  iR_VacuumAnalogMinDigit                   : UINT := 0;      (*Min value analog-input in digit*)
  iR_VacuumAnalogMaxDigit                   : UINT := 32737;  (*Max value analog-input in digit*)
  fR_VacuumAnalogMinMBar                    : REAL := 0;      (*Min value analog-input in mBar*)
  fR_VacuumAnalogMaxMBar                    : REAL := 50.0;   (*Max value analog-input in mBar*)
  fR_VacuumWarningLevelMBar                 : REAL := 20.0;   (*Warning level in mBar*)
  fR_VacuumErrorLevelMBar                   : REAL := 10.0;   (*Error level in mBar*)

  iR_ParticleMeasurementWarning             : INT := 40;      (*Particle measurement warning level*)
END_VAR

VAR CONSTANT
  iC_ParticleMeasurementNb                  : INT := 60;      (*Number of particle measurements*)
END_VAR

bO_FUReady := bI_FUReady;

fb_TofFUOffDelay(IN := bI_PrintActive, PT := tR_FUOffDelay);
bO_FUActivate := fb_TofFUOffDelay.Q;

fL_VacuumAnalogLevelMBar := UINT_TO_REAL(iI_VacuumMeasurement) * fR_VacuumAnalogMaxMBar / iR_VacuumAnalogMaxDigit;
  
fb_TonVacuumCheckDelay(IN := bO_FUActivate, PT := tR_VacuumCheckDelay);
IF fb_TonVacuumCheckDelay.Q THEN
  (*Level detection for messaging*)
  bO_VacuumWarningLevel := fL_VacuumAnalogLevelMBar < fR_VacuumWarningLevelMBar;
  bO_VacuumErrorLevel   := fL_VacuumAnalogLevelMBar < fR_VacuumErrorLevelMBar;
END_IF

AerosolMeasurement();

ACTION AerosolMeasurement:
fb_RTrigDataReceived(CLK := bI_AerosolMeasurementDataRec);
fb_FTrigDataReceived(CLK := bI_AerosolMeasurementDataRec);

CASE iL_COMstate OF
0:
  IF NOT bI_AerosolMeasurementAckInit THEN
    bO_AerosolMeasurementReqInit := TRUE;
  ELSE
    bO_AerosolMeasurementReqInit := FALSE;

    iL_COMstate := 1;

    bO_AerosolMeasurementAckRec := bI_AerosolMeasurementDataRec;
  END_IF

1:	(*Receive data*)
  IF    fb_RTrigDataReceived.Q
     OR fb_FTrigDataReceived.Q 
  THEN
    bO_AerosolMeasurementAckRec := bI_AerosolMeasurementDataRec;

    cL_Value := iI_AerosolMeasurementRecDataLength;

    aL_ReceivedData := '';
    FOR iL_Counter := 0 TO (cL_Value - 2) DO  (*Without Suffix*)
      aL_ReceivedData := CONCAT(aL_ReceivedData, F_ToCHR(cI_AerosolMeasurementRxBuff[iL_Counter]));
    END_FOR

    iL_ReceiveCount := iL_ReceiveCount + 1;
  END_IF

  IF    bI_AerosolMeasurementBufferFull
     OR bI_AerosolMeasurementFramingError
     OR bI_AerosolMeasurementOverRunError
  THEN
    iL_COMstate := 666;
  ELSE
    eO_ComState := eOpen;
  END_IF

666:	 (* ERROR STATE*)
  eO_ComState := ePortFaulty;	(*ERROR system*)
  iL_COMstate := 0;

END_CASE

fb_TonMeasurementTrigger(IN := NOT fb_TonMeasurementTrigger.Q, PT := T#10S);
IF fb_TonMeasurementTrigger.Q AND bO_FUActivate THEN
  fL_ParticleMeasurements[iL_ParticleMeasurementIdx] := fL_VacuumAnalogLevelMBar; (*TEST with fL_VacuumAnalogLevelMBar !!!*)
  iL_ParticleMeasurementIdx := iL_ParticleMeasurementIdx + 1;
  
  IF iL_ParticleMeasurementIdx > iC_ParticleMeasurementNb THEN
    FOR iL_Counter := 2 TO iC_ParticleMeasurementNb DO
      fL_ParticleMeasurements[iL_Counter - 1] := fL_ParticleMeasurements[iL_Counter];
    END_FOR
    iL_ParticleMeasurementIdx := iC_ParticleMeasurementNb;
  END_IF
END_IF
END_ACTION

METHOD mAckError : BOOL
VAR_INPUT
END_VAR
bO_VacuumWarningLevel := FALSE;
bO_VacuumErrorLevel   := FALSE;
END_METHOD

END_FUNCTION_BLOCK

// ---- POUs/Projects/Print/PRG_PRINT.TcPOU
PROGRAM PRG_PRINT
(*************************************************************************************************)
(*  FILENAME:    PRG_PRINT.EXP                                                                   *)
(*  PROJECT:     CALMAR PUPLC                                                                    *)
(*  COPYRIGHT:   All rights reserved (c) Wifag//Polytype, Fribourg/Switzerland (2016)            *)
(*  ENVIRONMENT: TwinCAT PLC                                                                     *)
(*  VERSION:     <version>                                                                       *)
(*************************************************************************************************)
(*  DESCRIPTION:                                                                   <description> *)
(*    Controls the digital print system.                                                         *)
(*    Main functions: start detection, printhead master, print unit, print group, print          *)
(*    controller.                                                                                *)
(*                                                                                </description> *)
(*************************************************************************************************)

VAR_INPUT
  (*EL5101*)
  lIKp_EncPulse                       AT%I* : ARRAY [1..iCPr_NB_PM] OF UDINT;       (*current encoder position*)
  bI_EncoderWcState                   AT%I* : ARRAY [1..iCPr_NB_PM] OF BOOL;        (*EL5101 encoder WcState*)
  
  bI_PuStopByInk                            : BOOL;  // PU stop and lock start from ink system
END_VAR

VAR_OUTPUT
  (*Interface OUT to PRG_INK / PRG_MACHINE*)
  bO_InitOk                                 : BOOL := FALSE;  (*Init Ok*)
  bO_PrintSystemOk                          : BOOL := TRUE;
  bO_TemperatureOk                          : BOOL := TRUE;
  bO_TotalWcState                           : BOOL := FALSE;  (*Monitoring: WcStates from all terminals*)
END_VAR

VAR
  nCtr, nCtr2 : UDINT;
  
  // ADS interface instances & mapping and responsible FBs
  // -------------------------------------------------------------
  FB_PU                                     : ARRAY [1..iCPr_NB_PU] OF FB_PU;               (*PU - Print Unit*)
  sAdsPrintUnit                             : ARRAY [1..iCPr_NB_PU] OF ST_ADS_PU;
  sL_BLK_PU                                 : ARRAY [1..iCPr_NB_PU] OF ST_MAP_BLK;
  sPuSettings                               : ST_PuSettings;                            // FB_PU configuration
  
  (*{attribute 'TcLinkTo' := '
    [1].fbPrintPosition.IlEncoderPulse := TIIB[RiGen5_v2]^Input^dsfsdfsa;
  '}*)
  fbPrintModule                             : ARRAY [1..iCPr_NB_PM] OF FB_PrintModule_WEU;
  sAdsPrintModule                           : ARRAY [1..iCPr_NB_PM] OF ST_ADS_PM;           (*PM -  Print Module *)
  sL_BLK_PM                                 : ARRAY [1..iCPr_NB_PM] OF ST_MAP_BLK;
//FB_PG                                     : ARRAY [1..iCPr_NB_PG] OF FB_PG;               (*PG -  Print Group *)
  sAdsPrintGroup                            : ARRAY [1..iCPr_NB_PG] OF ST_ADS_PG;
  sL_BLK_PG                                 : ARRAY [1..iCPr_NB_PG] OF ST_MAP_BLK;
  FB_PC                                     : ARRAY [1..iCPr_NB_PC] OF FB_PC;               (*PC - Print Controller*)
  sAdsPrintController                       : ARRAY [1..iCPr_NB_PC] OF ST_ADS_PC;
  sL_BLK_PC                                 : ARRAY [1..iCPr_NB_PC] OF ST_MAP_BLK;
  pFB_PC                                    : POINTER TO ARRAY [1..iCPr_NB_PC] OF POINTER TO FB_PC;
  //pFB_PC                                    : ARRAY [1..iCPr_NB_PC] OF POINTER TO FB_PC;    (* pointer array to PCs*)
  FB_PH                                     : ARRAY [1..iCPr_NB_PH] OF FB_PH_Grid;          (*PH - Print Head*)
  sAdsPrintHead                             : ARRAY [1..iCPr_NB_PH] OF ST_ADS_PH;
  sL_BLK_PH                                 : ARRAY [1..iCPr_NB_PH] OF ST_MAP_BLK;
  sAdsSheetAlignment                        : ARRAY [1..iCPr_NB_PU] OF ST_ADS_DVTSHEETALIGNMENT;          (*SA - Sheet alignement*)
  sL_BLK_SA                                 : ARRAY [1..iCPr_NB_PU] OF ST_MAP_BLK;
  sAdsSubstrate                             : ARRAY [1..iCPr_NB_SUBSTRATE_DEVICES] OF ST_ADS_SUBSTRATE;   (*SUB - Substrate*)
  sL_BLK_SUB                                : ARRAY [1..iCPr_NB_SUBSTRATE_DEVICES] OF ST_MAP_BLK;
  sAdsCamera                                : ARRAY [1..iCPr_NB_PU] OF ST_ADS_CAMERA;                     (*CAM - Camera*)  
  sL_BLK_CAMERA                             : ARRAY [1..iCPr_NB_PU] OF ST_MAP_BLK;          (*array of all camera blocks information*)
  // -------------------------------------------------------------

  // -------------------------------------------------------------
  // Configuration
  sC_Ads_Info                               : ST_ADS_INFO;      // PRG information for ADS block manager
  sMappingInfo                              : T_MapInfo;        // Block mapping configuration
  ISystemBase                               : I_SystemBase;     // reference to system base
  iSystemStatus                             : I_SystemStatus;   // System status interface
  //iSystemCmd                                : I_SystemCmd;      // System interface command
  
  pModuleDef                                : POINTER TO FB_ModuleDef;    // Module definition in system
  sC_Config_P                               : ST_CONFIG_P;      // PRG configuration  
  bL_InitRemVar                             : BOOL := TRUE;
  
  fbModuleMaster                            : FB_ModuleMaster;

  fbPm                                      : FB_ProdManager_DMAX;
  fbHardwarePool                            : FB_HardwarePool;
  fbDefGridParamMediator                    : FB_DefGridParamMediator;
     

  fbWorkerInspection                        : FB_WorkerDefGrid_Inspection;
  fbWorkerVerify                            : FB_WorkerDefGrid_Verify;
  fbWorkerDelete                            : FB_WorkerDefGrid_Delete;
  
  // globals
  rtPuStop                                  : R_TRIG;
  fbOd                                      : FB_OD;        // CoE object dictionary
  
  iWorker                                   : I_Worker;
  
  
  (* --- Maintainance variables ---*)
  (* - file download - *)
  (* -- fw/hw upgrade -- *)
  //fb_fwhw_update                            : FB_CALMAR_UPDATE;
	(* -- hib remote update -- *)
	//fb_pc_hib_rupd                            : ARRAY[1..iCPr_NB_PC] OF FB_PC_HIB_RUPD;(*HIB remote update channels*)
  //fb_hib_rup                                : FB_HIB_UPDATE;                         (*HIB remote updater*)
  (* -- stiching mask manager -- *)
  fb_fdl_mask                               : FB_FILE_DOWNLOAD;                      (*Mask file downloader*)
  (** -- waveform manager -- *)
  fb_fdl_waveform                           : FB_FILE_DOWNLOAD;                      (*waveform file downloader*)
  bWaveformDownloadErr                      : BOOL;                                  (*a waveform douwnload exitst (needed in RIGEN5 only)*)
  tOn_waveform                              : ARRAY[1..iCPr_NB_PC] OF TON;
  bL_waveform_request                       : ARRAY[1..iCPr_NB_PC] OF BOOL;
  lL_PhActStoragetankAssignmentIndex        : ARRAY[1..iCPr_NB_PH] OF DINT;
  lL_MemPhActStoragetankAssignmentIndex     : ARRAY[1..iCPr_NB_PH] OF DINT;
  
  

  
  
  
  
 (*----- Inspection System -----*)
  //bInspectionTrigger : BOOL;
  //fbInspectionSystemTrigger                 : FB_InspectionSystemTrigger;   // Inspection system trigger 
  //nInspectionSystemMarkIdx                  : INT := 3;

  // Neutral fibre calculation with additional mark sensors
  fbNeutralFibreDetermine                   : FB_NeutralFibreDetermine;    // Neutral fibre determine 
    
  (*----- Messages -----*)
  fb_Msg                                    : ARRAY [1..iC_NUM_MSG] OF FB_MESSAGE; (*global Module messages*)
  
  (* -- Recipe read/write auto-management*)
  pFbRecipeMngr                             : POINTER TO FB_RECIPE_READ_WRITE;
  
 
  
  (*----- print, offfset and motion variables ------*)
  // Trigger & Offsets
  //bL_StartTrigger                           : ARRAY [1..iCPr_NB_PM] OF BOOL;       (*Start Trigger for X0*)
  //rT_StartTrigger                           : ARRAY [1..iCPr_NB_PM] OF R_TRIG;
  nL_X0                                     : ARRAY [1..iCPr_NB_PM] OF DINT;       (*detected X0 position*)
  nL_X0_Comp                                : ARRAY [1..iCPr_NB_PM] OF DINT;       (*detected & adapted X0 start position*)
  nL_XS                                     : ARRAY [1..iCPr_NB_PG] OF DINT;       (*Shifted position of start print in pulse*)


  {warning 'TODO: refactor usage in PRG_INK'}
  stPcFlags                                 : ARRAY[1..iCPr_NB_PG] OF CalmarCompPrint.ST_PC_FLAGS;

  // Print module synchronisation
  //fbModuleSynchronisation                   : FB_ModuleSynchronisation;
  //bL_DisableModuleSynchronisation           : BOOL;   (*Visu: disable ModuleSynchronisation*)
  
  
  (*View*)
  // - VISU_SERVICE
  nServiceVisuFrameIndex                    : UINT := 0;   // VISU_SERVICE frame selection
  fbPrintOverview                           : FB_PrintOverview;
  
  (*Debug & Insight*)
  fbPrgPrintTest                            : FB_PrgPrint_test;
  LogPrSetup                                : T_NamedBase;  // just a I_LogSourceMacro implementation (logging PRINT module setup things)
  ePrint_LogLevel                           : E_LogSeverity  := E_LogSeverity.Debug;
  fbProfiler                                : FB_PrgProfiler;

  (*Simulation*)
  bSimulation                               : BOOL;
END_VAR
VAR CONSTANT
  (*Messaging*)
	iC_NUM_MSG                                : INT := 5;
	iC_MSG_1_FOE_MASK_ERR                     : INT := 1;
	iC_MSG_2_FOE_WAVEFORM_ERR                 : INT := 2;
  iC_MSG_3_FOE_CBFW_ERR                     : INT := 3;
  iC_MSG_4_FOE_HIBFW_ERR										: INT := 4;
  iC_MSG_5_PC_SUPPLY_OFF                    : INT := 5;
END_VAR

(* INIT First action init call*)
IF NOT bO_InitOk THEN
  Init();
  RETURN;
END_IF;

(* Call ACTIONS *)
(*************************************************************************************************)
RemVar();           (*Call update remanent data action*)
DownloadFiles();    (*Call file downloads*)
Testing();          (*Call test code*)
fbProfiler();
setLoggingLevels();


// Main/MasterModule part
fbModuleMaster();

// --------------------------------------------------------
// Print Blocks (global for all)
// -- CT and ProdMngr (Production Management)


fbOd();
fbPm();
fbHardwarePool();


// -- PM print modules
FOR nCtr := 1 TO TO_UDINT(iCPr_NB_PM) DO
  
  FOR nCtr2 := 1 TO TO_UDINT(GVL_WEU.nC_WorkerPrintPerPm) DO
    {warning 'TODO: scale X Offset with fL_WebStretchCalculated?'}
    fbPrintModule[nCtr].fPrintOffsetX[nCtr2]       :=  TO_LREAL(sAdsPrintUnit[ePr_PU_UNIT_1].sI_ShiftJobX.lI_Val) / 1_000_000 	// PU [um] to [m]
                                                     + TO_LREAL(sAdsPrintModule[nCtr].sI_GeneralShiftX.lI_Val) / 1_000_000 	  // PG [um] to [m]
                                                     + TO_LREAL(sAdsPrintGroup[nCtr2 + TO_UDINT(iCPr_MAP_PM_PG[nCtr2])-1].sI_ShiftPositionX.lI_Val) / 1_000_000;
    fbPrintModule[nCtr].fPrintOffsetY[nCtr2]       :=  DINT_TO_LREAL(F_MeterToSubPixel(DINT_TO_LREAL(sAdsPrintUnit[ePr_PU_UNIT_1].sI_ShiftJobY.lI_Val ) / 1_000_000, nC_PrintResolution))   (*[um] to [px] job yOffset from upper level (GUI)*)
                                                     + DINT_TO_LREAL(F_MeterToSubPixel(DINT_TO_LREAL(sAdsPrintModule[nCtr].sI_GeneralShiftY.lI_Val )    / 1_000_000, nC_PrintResolution))   (*[um] to [px] job yOffset from upper level (GUI)*)
                                                     + DINT_TO_LREAL(F_MeterToSubPixel(DINT_TO_LREAL(sAdsPrintGroup[nCtr2 + TO_UDINT(iCPr_MAP_PM_PG[nCtr2])-1].sI_ShiftPositionY.lI_Val) / 1_000_000, nC_PrintResolution));   (*[um] to [px] job yOffset from upper level (GUI)*)
                                                      
	END_FOR
    
  fbPrintModule[nCtr]();
END_FOR



// Print module synchronisation (simulation not for production)
(*
fbModuleSynchronisation( IbEnable           := NOT bL_DisableModuleSynchronisation
                       , IbEngaged          := bL_Engaged
                       , IbPrintEnabled     := bL_PrintEnabled
                       , InFormatLength     := nL_FormatLength
                       , InModule2ToModule3 := nL_Module2ToModule3
                       , IbFormatTrig       := bL_StartTrig
                       , ObPrintEnabled     => bL_PrintEnabledSync); 
*)


// --------------------------------------------------------
// Worker chain  --> call all work() methods
iWorker := fbWorkerDelete.Root;
WHILE iWorker <> 0 DO
  iWorker.work();
  iWorker := iWorker.Next;
END_WHILE


(* -- PU PrintUnit*)
// PG->PU status/flags 
FOR nCtr := 1 TO TO_UDINT(iCPr_NB_PU) DO 
  // specific handling
  rtPuStop(CLK := bI_PuStopByInk);       (*If varnish change is activated the job should be stopped.*)
  IF rtPuStop.Q THEN FB_PU[nCtr].reqPuStop('Stop by InkSystem'); END_IF
  
  FB_PU[nCtr]();
  
  // WEU Start CanEx override
  sAdsPrintUnit[nCtr].sI_Start.bO_CommandCanEx := sAdsPrintUnit[nCtr].sI_Start.bO_CommandCanEx 
                                                AND NOT iSystemStatus.bSleep     // sleep active
                                                AND NOT bI_PuStopByInk;          // ink system locks start
END_FOR

// Inspection system
{warning 'TODO: create a worker for inspection system'}
(*
IF (nInspectionSystemMarkIdx > 3) OR (nInspectionSystemMarkIdx < 2) THEN nInspectionSystemMarkIdx := 3; END_IF  (*Index check*)
fbInspectionSystemTrigger.UsePositionTrigger := fbStartPositionSimulationHOA._bSim AND NOT bL_DisableSimMarkStartTriggerM3;
(*input bI_SensorState depends on _bUsePositionTrigger*)
IF fbInspectionSystemTrigger.UsePositionTrigger THEN
  fbInspectionSystemTrigger.bI_SensorState := bMasterTrigger;
ELSE
  fbInspectionSystemTrigger.bI_SensorState := Fb_PaperPosDetect[nInspectionSystemMarkIdx - 1].bIKp_StartSensor;
END_IF

fbInspectionSystemTrigger.bI_SensorState
fbInspectionSystemTrigger( iI_CurrentPos         := nMasterPosition
                         , fI_ConveyorSpeed      := fMasterSpeed
                         , iI_SensorX0           := SEL(bL_Engaged[1], nL_X0[2]                           , nL_X0[1])
                         , tI_SensorTimeStampPos := Fb_PaperPosDetect[nInspectionSystemMarkIdx - 1].tIKp_TimeStampPos
                         (*StartTrigger Simulation VISU&FB*)
                       //, bI_ManualTrigger      := fbStartPositionSimulation.bStartTrig
                         );
*)

// Neutral fibre calculation with additional mark sensors
fbNeutralFibreDetermine(fSpeed := fbModuleMaster.fMasterSpeed);


(*--- VISU stuff ----------------*)
// fix offset (left visu border) + VerifyWorker = a constant position => calculate a pixel to m ratio
fbPrintOverview.fX_m  := fbWorkerDelete.fPosition; // (0.2 + fbWorkerVerify.fWorkerToMasterRef) + fbModuleMaster.fLastModuleOffset + (fbModuleMaster.fDetectToRefPos);
fbPrintOverview.fY_m  := 2;
fbPrintOverview.nX_px := 800;
fbPrintOverview.nY_px := 300;
fbPrintOverview.fPxToMRatio := fbPrintOverview.nX_px / fbPrintOverview.fX_m;
fbPrintOverview.iPrintPosition := fbModuleMaster.iMasterPrintPosition;

fbPrintOverview();
(*------------------------------*)

(****************************************************************************)
(* Messaging, NOTE: they are using the FB_PU message handler! *)
(* ------------------------------------------------------------------------ *)
fb_Msg[iC_MSG_1_FOE_MASK_ERR]    .bI_Status := fb_fdl_mask.bO_Error;
fb_Msg[iC_MSG_2_FOE_WAVEFORM_ERR].bI_Status := FALSE;  //bWaveformDownloadErr; // fb_fdl_waveform.bO_Error;
fb_Msg[iC_MSG_3_FOE_CBFW_ERR]    .bI_Status := fbHardwarePool.bError_fwhw_update;
fb_Msg[iC_MSG_4_FOE_HIBFW_ERR]   .bI_Status := fbHardwarePool.bError_hib_rup;
fb_Msg[iC_MSG_5_PC_SUPPLY_OFF]   .bI_Status := FALSE; //TODO: NOT PRG_MACHINE.sL_CvyrStatus.bI_PowerState;

FOR nCtr := 1 TO TO_UDINT(iC_NUM_MSG) DO
  IF fb_Msg[nCtr].pI_MsgConfig <> 0 AND fb_Msg[nCtr].iI_MsgNumber <> 0 THEN
    fb_Msg[nCtr]();
  END_IF
END_FOR 

(****************************************************************************)
(* Global states *)
(* ------------------------------------------------------------------------ *)
bO_PrintSystemOk := fbPm.bReady;
(*WcState: 0 = Data valid, 1 = Data invalid*)
bO_TotalWcState :=    bI_EncoderWcState[1]
                   OR bI_EncoderWcState[2];

METHOD DownloadFiles
VAR
  lCtr : INT;
  sPcFlags : ST_PC_FLAGS;
  aDefaultWaveform : T_MaxString;
  aInkWaveform : T_MaxString;
END_VAR
(* PC firmware updater*)
(*    uses PC[x] FoE channel *)
(* ------------------------------------------------------------------------ *)
(* --- START: --- *)
//fb_fwhw_update( pI_fbPc := pFB_PC^);
(* --- END: --- *)


(****************************************************************************)
(* HIB remote update*)
(*    uses PC[x] FoE channel *)
(* ------------------------------------------------------------------------ *)
(* --- START: --- *)
//fb_hib_rup();
(* --- END: --- *)


(****************************************************************************)
(* mask update*)
(*		uses PC[x] FoE channel *)
(* ------------------------------------------------------------------------ *)
(* --- START: printhead mask loader --- *)
(*FOR lCtr := 1 TO iCPr_NB_PC DO
  IF FB_PC[lCtr].sO_PcFlags.bBoardEnterOp THEN 
    fb_fdl_mask.Start(DINT_TO_INT(lCtr));    // start individual channel
	END_IF
END_FOR;*)
fb_fdl_mask();
(* --- END: printhead mask loader --- *)


(****************************************************************************)
(* Waveform update*)
(*    uses PC[x] FoE channel *)
(* ------------------------------------------------------------------------ *)
(* --- START: printhead waveform loader --- *)
bWaveformDownloadErr := FALSE;
FOR lCtr := 1 TO iCPr_NB_PC DO
  sPcFlags := FB_PC[lCtr].sPcFlags;
  bL_waveform_request[lCtr] := tOn_waveform[lCtr].Q;
  IF    ( sPcFlags.bBoardEnabling ) 
     OR ( bL_waveform_request[lCtr] ) //filtered internally: AND NOT fb_fdl_waveform[iL_Counter].bO_Busy AND (tTimeoutWavef[iL_Counter].Q OR fb_Wavef_CfgTrig[iL_Counter].Q)
  THEN
    fb_fdl_waveform.Start(DINT_TO_INT(lCtr));    // start individual channel
  END_IF

  tOn_waveform[lCtr](IN:=sPcFlags.bWaveform AND NOT bL_waveform_request[lCtr], PT:= T#14S);

  // build global request for message
  IF sPcFlags.bWaveform AND FB_PC[lCtr].bBoardEnable THEN 
    bWaveformDownloadErr := TRUE;
	END_IF
END_FOR;
fb_fdl_waveform();

(*Assign WaveFileName from storage tank to PH. Trigger transmit of waveform if new name is set.*)
FOR lCtr := 1 TO iCPr_NB_PH DO
  lL_PhActStoragetankAssignmentIndex[lCtr] := PRG_INK.iL_ActStoragetankAssignmentIndex[iCPr_MAP_PH_HT[lCtr]];

  (*If lL_PhActStoragetankAssignmentIndex is assigned to a storage tank the waveform must be copied.*)
  IF     (lL_PhActStoragetankAssignmentIndex[lCtr] > 0)
     AND (lL_PhActStoragetankAssignmentIndex[lCtr] <> lL_MemPhActStoragetankAssignmentIndex[lCtr])
  THEN
    // set new waveform name to PH
    aDefaultWaveform := fb_fdl_waveform.aI_src_file_name_default;
    aInkWaveform := PRG_INK.sAdsIkInkStorageTank[lL_PhActStoragetankAssignmentIndex[lCtr]].sI_InkParameter.aWaveform; 
    
    IF aInkWaveform <> '' AND aInkWaveform <> 'undef' AND aInkWaveform <> 'undef.wav' THEN  // use only when waveform from storage assignemen is ok, else keep ph ads value
      sAdsPrintHead[lCtr].aI_WaveFileName := PRG_INK.sAdsIkInkStorageTank[lL_PhActStoragetankAssignmentIndex[lCtr]].sI_InkParameter.aWaveform;      
		END_IF

    (*Fix extension if not existing in the file name*)
    IF (FIND(sAdsPrintHead[lCtr].aI_WaveFileName, '.wav') = 0) AND (FIND(sAdsPrintHead[lCtr].aI_WaveFileName, '.WAV') = 0) THEN
      sAdsPrintHead[lCtr].aI_WaveFileName := CONCAT(sAdsPrintHead[lCtr].aI_WaveFileName, '.wav');
    END_IF

    (*check for valid file name*)
     IF sAdsPrintHead[lCtr].aI_WaveFileName = 'undef.wav' OR sAdsPrintHead[lCtr].aI_WaveFileName = '.wav' OR sAdsPrintHead[lCtr].aI_WaveFileName = '' THEN
       LogPrSetup.LogError(F_Concat5('Invalid waveform filename: ', sAdsPrintHead[lCtr].aI_WaveFileName, ' on PH[', TO_STRING(lCtr),']'));
       sAdsPrintHead[lCtr].aI_WaveFileName := aDefaultWaveform;
       LogPrSetup.LogError(F_Concat5('Set default waveform filename: ', sAdsPrintHead[lCtr].aI_WaveFileName, ' on PH[', TO_STRING(lCtr),']'));
		 END_IF
  END_IF

  lL_MemPhActStoragetankAssignmentIndex[lCtr] := lL_PhActStoragetankAssignmentIndex[lCtr];
END_FOR
END_METHOD

METHOD Init : BOOL
VAR
  nCtr : UDINT;
  nPhCtr : UDINT;
  pAdsPg : ARRAY[1..GVL_WEU.nC_WorkerPrintPerPm] OF POINTER TO ST_ADS_PG;
END_VAR
(*************************************************************************************************)
(* --- Module preprarations --- *)

// Get system reference
IF ISystemBase = 0 THEN
  ISystemBase := PRG_SYSTEMBASE.getSystemBaseInterface();
  IF ISystemBase = 0 THEN 
    RETURN; 
  END_IF
END_IF

// Wait until system(base) is booted
IF ISystemBase.bBooting THEN RETURN; END_IF
PRG_SYSTEMBASE.getSystemStatusInterface(iSystemStatus=>iSystemStatus);
//PRG_SYSTEMBASE.getSystemCmdInterface(iSystemCmd=>iSystemCmd

// Build mapping information for ADS
Mapping();

// Register module to system
pModuleDef := ISystemBase.regModule(
  pAdsInfo := ADR(sC_Ads_Info),
  pMapInfo := ADR(sMappingInfo)
);
IF pModuleDef = 0 THEN RETURN; END_IF

// remanent init 
RemVar();



(*************************************************************************************************)
(* Init FB and ADS instances*)
setLoggingLevels();

(*-- Print blocks init --------------------------------------------------------------------------*)
(*-- Module Master*)
fbModuleMaster.Init(pPU:=ADR(FB_PU[1]), pProdMngr:=ADR(fbpm), iHwPool:=fbHardwarePool);


(*-- CoE object dicionary*)
fbOd.init(aAmsNetId:=sC_AMSNETID_LOCALHOST, aFilePath:=F_Concat3(aC_PlcConfigPath, aC_PlcFlashFileSubPath, 'od.json'), pSimString:=0);

(* -- PU PrintUnit*)
FOR nCtr := 1 TO TO_UDINT(iCPr_NB_PU) DO
	(*-- ADS --*)
  setupAdsPu(pAds:=ADR(sAdsPrintUnit[nCtr]), nIdx:=nCtr);
  setupAdsSa(pAds:=ADR(sAdsSheetAlignment[nCtr]));
  
	(*-- FB --*)
  sPuSettings.bStopAfterDone := FALSE;
  FB_PU[nCtr].Init(                                                  (*Init referenced & config for FB*)
                    pAdsIf        := ADR(sAdsPrintUnit[nCtr])        (*> ads pu reference*)
                  , pAdsSubstrate := ADR(sAdsSubstrate[1])           (*> ads substrate ref*)
                  , pPuSettings   := ADR(sPuSettings)
                  , iNumPg        := iCPr_NB_PM                      (*> Number print SubSystems*)
                  );
END_FOR;


(* -- PG PrintGroup*)
FOR nCtr := 1 TO TO_UDINT(iCPr_NB_PG) DO
	(*-- ADS --*)
  setupAdsPg(pAds:=ADR(sAdsPrintGroup[nCtr]), nIdx:=nCtr);

  (*-- IF direct access to PRG_INK --*)
  PRG_INK.pAdsPg[nCtr] := ADR(sAdsPrintGroup[nCtr]);  
END_FOR;


// !!! Init HW before module (PCs, PHs) !!! --------------------
(* -- PC Print Controller*)
FOR nCtr := 1 TO TO_UDINT(iCPr_NB_PC) DO
	(*-- PC --*)
	FB_PC[nCtr].Init( pAds               := ADR(sAdsPrintController[nCtr])
                  , sAmsNetIdLocalHost := sC_AMSNETID_LOCALHOST
                  , sAmsNetIdIo        := sC_AMSNETID_IO
                  , nEcatSlaveAddr     := iG_PC_ADDRESS[nCtr]
                  , nBlockId           := ePr_BLK_PC
                  , pOd                := ADR(fbOd)
                  , tWaveDownload      := T#10S
                  );
  
  // hw enable inputs not existing -> enable initially
  FOR nPhCtr := 1 TO TO_UDINT(iCPr_NB_PH_PER_CONTROLLER) DO
    FB_PC[nCtr].bI_PhHwEnable[nPhCtr] := TRUE;
  END_FOR

	(*-- ADS --*)
  setupAdsPc(pAds:=ADR(sAdsPrintController[nCtr]), nIdx:=nCtr);
END_FOR;


(*PH - Print Head*)
FOR nCtr := 1 TO TO_UDINT(iCPr_NB_PH) DO
	(*-- ADS --*)
  setupAdsPh(pAds:=ADR(sAdsPrintHead[nCtr]), nIdx:=nCtr);
     
  fbPrintModule[iCPr_PH_MAPPING[nCtr].nPm].RegisterHw(
    pPc:=ADR(FB_PC[iCPr_PH_MAPPING[nCtr].nPcInst]),
    pPh:=ADR(FB_PH[iCPr_PH_MAPPING[nCtr].nPhInst]),
    pMapDef:=ADR(iCPr_PH_MAPPING[nCtr])
  );

  (*-- PH --*)
  FB_PH[nCtr].init( pAdsIf       := ADR(sAdsPrintHead[nCtr])
                  , sPhDef       := GVL_PrintDef.RIGEN5
                  , tTempMonitor := T#45S
                  );
END_FOR;


(*----SUBSTRATE init*)
FOR nCtr := 1 TO TO_UDINT(iCPr_NB_SUBSTRATE_DEVICES) DO
  setupAdsSub(pAds:=ADR(sAdsSubstrate[nCtr]), nIdx:=nCtr); 
END_FOR


(*-- PrintModules*)
FOR nCtr := 1 TO TO_UDINT(iCPr_NB_PM) DO

	(*-- ADS --*)
  setupAdsPm(pAds:=ADR(sAdsPrintModule[nCtr]), nIdx:=nCtr);
  
  pAdsPg[1] := ADR(sAdsPrintGroup[iCPr_MAP_PM_PG[nCtr]]);
  pAdsPg[2] := ADR(sAdsPrintGroup[iCPr_MAP_PM_PG[nCtr]+1]);
  
  (*-- FB -- *)
  {warning 'TODO: set size: fPrintUnitWidth'}
  fbPrintModule[nCtr].Init( nIdx     := TO_UDINT(nCtr)
                          , pAdsPm   := ADR(sAdsPrintModule[nCtr])
                          , pAdsSa   := ADR(sAdsSheetAlignment[ePr_PU_UNIT_1])
                          , pAdsCam  := ADR(sAdsCamera[1])
                          , pAdsPg   := pAdsPg
                          , fCycleTime := pModuleDef^.fCycleTime_s
                          , fPrintUnitWidth := 1  {warning 'TODO: used for Grid ImageShift somehow and banana correction'}
                          , nYShiftPcCenter := nC_YShiftOffset
                          , iModuleMaster := fbModuleMaster
                          , iPosition := 0  // set internally
                          , iStartPos := 0  // set internally
                          , iSystemStatus := iSystemStatus
                          , pMachineInputs := ADR(PRG_MACHINE.fbMachineComm.sModuleMachineState[nCtr])
                          , pMachineOutputs := ADR(PRG_MACHINE.fbMachineComm.sModuleMachineFeedback[nCtr])
  );
  // register to master
  fbModuleMaster.registerModule(pModule:=ADR(fbPrintModule[nCtr]));
END_FOR;
fbModuleMaster.setMasterModule(ADR(fbPrintModule[1]));


(*-- Print management init ------------------------------------------------------------------*)
fbPm.LogLevel := ePrint_LogLevel;
fbPm.init( pPU    := ADR(FB_PU[ePr_PU_UNIT_1]) 
         , pAdsPU := ADR(sAdsPrintUnit[ePr_PU_UNIT_1]),
         );
fbPm();  // call it once for self-initialisation
FB_PU[ePr_PU_UNIT_1].registerStatusClient(sClient := fbPm);


(*-- Worker init --------------------------------------------------------------------------------*)


// -- Worker Print
//  -> defined in Module

// -- Verify
fbWorkerVerify.Init(iWorkerParams:=fbModuleMaster.iWorkerParams, pMsgConfig:=FB_PU[1].pO_MsgConfig, fPrintResolution := nC_PrintResolution, fSubPxResolution := nC_SubPixelResolution);
fbWorkerVerify.InitWorkerVerify(pPm:=ADR(fbPm));
fbWorkerVerify.reg();
fB_PU[ePr_PU_UNIT_1].registerStatusClient(sClient:=fbWorkerVerify);

// -- Inspection
fbWorkerInspection.Init(iWorkerParams:=fbModuleMaster.iWorkerParams, pMsgConfig:=FB_PU[1].pO_MsgConfig, fPrintResolution := nC_PrintResolution, fSubPxResolution := nC_SubPixelResolution);
fbWorkerInspection.reg();
fB_PU[ePr_PU_UNIT_1].registerStatusClient(sClient:=fbWorkerInspection);

// -- Delete
fbWorkerDelete.Init(iWorkerParams:=fbModuleMaster.iWorkerParams, pMsgConfig:=FB_PU[1].pO_MsgConfig, fPrintResolution := nC_PrintResolution, fSubPxResolution := nC_SubPixelResolution);
fbWorkerDelete.reg();
fB_PU[ePr_PU_UNIT_1].registerStatusClient(sClient:=fbWorkerDelete);


(*-- Camera init ----------------------------------------------------*)

// -- No camera (SheetDetect only)
//fbNoCamera.Init(nPrintUnitResolution:=nC_PrintResolution, nPrintUnitSubPx:=nC_SubPixelResolution, iCameraTrigger:=fbMarkDetection, bUseCameraTrigger:=FALSE, bUseCameraTriggerFeedback:=FALSE);
//fbWorkerCamera.RegisterCamera(fbNoCamera);


// -- Param mediator between Workers
//fbDefGridParamMediator.init(pCreateWorker:=ADR(fbWorkerDefGrid_Python), pCamWorker := ADR(fbWorkerDefGrid_Camera),pDefWorker:= ADR(fbWorkerDefGrid_Deformation));

// register Emergency
(*FOR lCtr := 1 TO iCPr_NB_PG DO
  PRG_SYSTEMBASE.fbEmergency.mRegisterObserver(iObserver := fbWorkerWeu[lCtr]);
END_FOR*)


// Hw Management
//    Hardware Pool for PH - Print Head and PC - Print Controller*)
fBHardwarePool.init(
  sAmsNetIdLocalhost  := sC_AMSNETID_LOCALHOST,
  sAmsNetIdIo         := sC_AMSNETID_IO,
  pOd                 := ADR(fbOd),
  pConfig             := ADR(sC_Config_P)
);
pFB_PC := fbHardwarePool.pPcs;  // used for FileDownload and global FBs managing all PCs




(*************************************************************************************************)
(*FileDownloader*)

//(* - firmware*) - Is now in HardwarePool
//fb_fwhw_update.aI_appl_file_path := F_Concat3(aC_PlcConfigPath, aC_PlcFlashFileSubPath, 'user.appl');
//fb_fwhw_update.aI_fpga_file_path := F_Concat3(aC_PlcConfigPath, aC_PlcFlashFileSubPath, 'user.fpga');
//fb_fwhw_update( pI_fbPc := pFB_PC^);
//fb_fwhw_update.init();

//(* - hib remote upfate*) - Is now in HardwarePool
//fb_hib_rup.bI_Enable   := TRUE;
//fb_hib_rup.aI_FilePath := F_Concat3(aC_PlcConfigPath, aC_PlcFlashFileSubPath, 'user.hib');
//fb_hib_rup( sI_Ary_Fb:=fb_pc_hib_rupd, pI_Ary_Fb_Pc:=pFB_PC^);


(*-- Mask file*)
fb_fdl_mask.bI_Enable                := TRUE;
fb_fdl_mask.aI_src_file_path         := CONCAT(aC_PlcConfigPath, aC_PlcMaskFileSubPath);
fb_fdl_mask.aI_src_file_name_default := 'mask.msk';
fb_fdl_mask.aI_dest_file_path        := 'mask.msk.msk';
FOR nCtr := 1 TO TO_UDINT(iCPr_NB_PC) DO
	FOR nPhCtr := 1 TO TO_UDINT(iCPr_NB_PH_PER_CONTROLLER) DO
		IF iCPr_MAP_PC_PH[nCtr, nPhCtr] <> -1 THEN
	    fb_fdl_mask.aI_src_file_names[nCtr, nPhCtr] := ADR(sAdsPrintHead[iCPr_MAP_PC_PH[nCtr, nPhCtr]].aI_MaskFileName);
		END_IF
	END_FOR
END_FOR
fb_fdl_mask(pI_fbpc:=pFB_PC^);
fb_fdl_mask.Init(
  aDownloaderName := 'Mask downloader',
  bFilePerPh      := TRUE,
  bDefaultFile    := FALSE,
  bShowDetail     := TRUE,
  bUseLock        := FALSE,
  bEnabledOnly    := TRUE,
  bFileNameChange := TRUE,
  bEnterOp        := TRUE,
  bEnabling       := TRUE,
  bUseRange       := FALSE,
  lColorRGB       := 16#FF0080FF,
  iRetryCount     := 0,
  tRetryTimeout   := T#8S,
);

(*-- waveform file*)
fb_fdl_waveform.bI_Enable                := TRUE;
fb_fdl_waveform.aI_src_file_path         := CONCAT(aC_PlcConfigPath, aC_PlcWaveformFileSubPath);
fb_fdl_waveform.aI_src_file_name_default := 'waveform.wav';
fb_fdl_waveform.aI_dest_file_path        := 'waveform.wav.wav';
FOR nCtr := 1 TO TO_UDINT(iCPr_NB_PC) DO
	FOR nPhCtr := 1 TO TO_UDINT(iCPr_NB_PH_PER_CONTROLLER) DO
		IF iCPr_MAP_PC_PH[nCtr, nPhCtr] <> -1 THEN
	    fb_fdl_waveform.aI_src_file_names[nCtr, nPhCtr] := ADR(sAdsPrintHead[iCPr_MAP_PC_PH[nCtr, nPhCtr]].aI_WaveFileName);
		END_IF
	END_FOR
END_FOR
fb_fdl_waveform(pI_fbpc:=pFB_PC^);
fb_fdl_waveform.Init(
  aDownloaderName := 'Waveform downloader',
  bFilePerPh      := FALSE,
  bDefaultFile    := FALSE,
  bShowDetail     := TRUE,
  bUseLock        := FALSE,
  bEnabledOnly    := TRUE,
  bFileNameChange := TRUE,
  bEnterOp        := TRUE,
  bEnabling       := TRUE,
  bUseRange       := FALSE,
  lColorRGB       := 16#FF9191C8,
  iRetryCount     := 0,
  tRetryTimeout   := T#9S,  
);


// View setup
fbPrintOverview.init(
  pCTM:=fbModuleMaster.pCTManager, 
  pWorkerDefGrid:=ADR(fbWorkerDelete)
);

// Inspection system
//fbInspectionSystemTrigger.Init(nResolution := nC_PrintResolution * nC_SubPixelResolution, bUsePositionTrigger := FALSE);

// Neutral fibre calculation with additional mark sensors
fbNeutralFibreDetermine.Init(nResolution := nC_PrintResolution * nC_SubPixelResolution);


(*Messaging*)
(*************************************************************************************************)
(*NOTE: FB_PU[x].init() has to be called before*)
fb_Msg[iC_MSG_1_FOE_MASK_ERR].pI_MsgConfig       := FB_PU[1].pO_MsgConfig;
fb_Msg[iC_MSG_1_FOE_MASK_ERR].iI_MsgLocation     := ePr_BLK_PU;
fb_Msg[iC_MSG_1_FOE_MASK_ERR].iI_MsgNumber       := eCPr_FOE_MASK_DL_ERR;

fb_Msg[iC_MSG_2_FOE_WAVEFORM_ERR].pI_MsgConfig   := FB_PU[1].pO_MsgConfig;
fb_Msg[iC_MSG_2_FOE_WAVEFORM_ERR].iI_MsgLocation := ePr_BLK_PU;
fb_Msg[iC_MSG_2_FOE_WAVEFORM_ERR].iI_MsgNumber   := eCPr_FOE_WAVEFORM_DL_ERR;

fb_Msg[iC_MSG_3_FOE_CBFW_ERR].pI_MsgConfig       := FB_PU[1].pO_MsgConfig;
fb_Msg[iC_MSG_3_FOE_CBFW_ERR].iI_MsgLocation     := ePr_BLK_PU;
fb_Msg[iC_MSG_3_FOE_CBFW_ERR].iI_MsgNumber       := eCPr_FOE_CBFW_DL_ERR;

fb_Msg[iC_MSG_4_FOE_HIBFW_ERR].pI_MsgConfig      := FB_PU[1].pO_MsgConfig;
fb_Msg[iC_MSG_4_FOE_HIBFW_ERR].iI_MsgLocation    := ePr_BLK_PU;
fb_Msg[iC_MSG_4_FOE_HIBFW_ERR].iI_MsgNumber      := eCPr_FOE_HIBFW_DL_ERR;

fb_Msg[iC_MSG_5_PC_SUPPLY_OFF].pI_MsgConfig      := FB_PU[1].pO_MsgConfig;
fb_Msg[iC_MSG_5_PC_SUPPLY_OFF].iI_MsgLocation    := ePr_BLK_PU;
fb_Msg[iC_MSG_5_PC_SUPPLY_OFF].iI_MsgNumber      := eCPr_PC_SUPPLY_OFF;


(*************************************************************************************************)
(* --- System servcices ---- *)
(* -- BlockId saving ----------------------------------------------------------------------------*)
PRG_SYSTEMBASE.fbBlockIdSave.registerModule(
  aI_StoragePath := CONCAT(aC_PlcConfigPath, aC_PlcBlockIdSubPath),
  pI_Ads_Info    := ADR(sC_Ads_Info)
);

// init finished
bO_InitOk := TRUE;

(**** END ****************************************************************************************)
END_METHOD

METHOD Mapping : BOOL
VAR
  lCtr : INT;
END_VAR
(*************************************************************************************************)
(*ADS blocks mapping definition*)
(*************************************************************************************************)
(*mapping of each block with his parents, type and index*)
(*unit -> root*)
sL_BLK_PU[1].iPMaps[1]    := FC_ADD_MAP(eSys_BLK_ROOT, 1);

(*Substrate -> root*)
sL_BLK_SUB[1].iPMaps[1]   := FC_ADD_MAP(eSys_BLK_ROOT, 1);

(*SheetAlignment -> unit*)
sL_BLK_SA[1].iPMaps[1]    := FC_ADD_MAP(ePr_BLK_PU, 1);

(*Camera -> unit*)
sL_BLK_CAMERA[1].iPMaps[1]:= FC_ADD_MAP(ePr_BLK_PU, 1);

(*module*)
FOR lCtr := 1 TO iCPr_NB_PM DO
  (*modules -> unit*)
  sL_BLK_PM[lCtr].iPMaps[1] := FC_ADD_MAP(ePr_BLK_PU, 1);
END_FOR;

(*group*)
FOR lCtr := 1 TO iCPr_NB_PG DO
  (*groups -> module*)
  sL_BLK_PG[lCtr].iPMaps[1] := FC_ADD_MAP(ePr_BLK_PM, iCPr_MAP_PG_PM[lCtr]);
  (*groups -> header tank group*)
  sL_BLK_PG[lCtr].iPMaps[2] := FC_ADD_MAP(eIk_BLK_HEADERTANK_GROUP, iCPr_MAP_PG_HTG[lCtr]);
END_FOR;

(*controller*)
FOR lCtr := 1 TO iCPr_NB_PC DO
  (*controller -> group*)
  IF bCPr_PC_EXIST[lCtr] THEN
    sL_BLK_PC[lCtr].iPMaps[1] := FC_ADD_MAP(ePr_BLK_PG, iCPr_MAP_PC_PG[lCtr]);
  END_IF;
END_FOR;

(*printhead*)
FOR lCtr := 1 TO iCPr_NB_PH DO
  (*printhead -> print controller*)
  IF bCPr_PH_EXIST[lCtr] THEN
    sL_BLK_PH[lCtr].iPMaps[1] := FC_ADD_MAP(ePr_BLK_PC        , iCPr_MAP_PH_PC[lCtr]);
  END_IF;
END_FOR;


(*************************************************************************************************)
(* initialize module information (module and mapping) *)
(*************************************************************************************************)
sC_Ads_Info.bReady   := FALSE;
sC_Ads_Info.aType    := 'PRG_PRINT';
sC_Ads_Info.iVersion := 010000;			(*1.0.0*)
sC_Ads_Info.iType    := eMOD_PRINT;

sMappingInfo.init(lModId:=TO_UINT(eMOD_PRINT));
sMappingInfo.addBlkAry( iAdsBlockType := TO_UINT(ePr_BLK_PU),       aAdsBlockName := 'sAdsPrintUnit',       iAdsBlockVersion:= sAdsPrintUnit[1].iO_Version,                    iNbrBlocks := SIZEOF(sL_BLK_PU)/SIZEOF(sL_BLK_PU[1]),         pBlockArray := ADR(sL_BLK_PU));
sMappingInfo.addBlkAry( iAdsBlockType := TO_UINT(ePr_BLK_PM),       aAdsBlockName := 'sAdsPrintModule',     iAdsBlockVersion:= INT_TO_UINT(sAdsPrintModule[1].iO_Version),     iNbrBlocks := SIZEOF(sL_BLK_PM)/SIZEOF(sL_BLK_PM[1]),         pBlockArray := ADR(sL_BLK_PM));
sMappingInfo.addBlkAry( iAdsBlockType := TO_UINT(ePr_BLK_PG),       aAdsBlockName := 'sAdsPrintGroup',      iAdsBlockVersion:= INT_TO_UINT(sAdsPrintGroup[1].iO_Version),      iNbrBlocks := SIZEOF(sL_BLK_PG)/SIZEOF(sL_BLK_PG[1]),         pBlockArray := ADR(sL_BLK_PG));
sMappingInfo.addBlkAry( iAdsBlockType := TO_UINT(ePr_BLK_PC),       aAdsBlockName := 'sAdsPrintController', iAdsBlockVersion:= INT_TO_UINT(sAdsPrintController[1].iO_Version), iNbrBlocks := SIZEOF(sL_BLK_PC)/SIZEOF(sL_BLK_PC[1]),         pBlockArray := ADR(sL_BLK_PC));
sMappingInfo.addBlkAry( iAdsBlockType := TO_UINT(ePr_BLK_PH),       aAdsBlockName := 'sAdsPrintHead',       iAdsBlockVersion:= INT_TO_UINT(sAdsPrintHead[1].iO_Version),       iNbrBlocks := SIZEOF(sL_BLK_PH)/SIZEOF(sL_BLK_PH[1]),         pBlockArray := ADR(sL_BLK_PH));
sMappingInfo.addBlkAry( iAdsBlockType := TO_UINT(ePr_BLK_SA),       aAdsBlockName := 'sAdsSheetAlignment',  iAdsBlockVersion:= INT_TO_UINT(sAdsSheetAlignment[1].iO_Version),  iNbrBlocks := SIZEOF(sL_BLK_SA)/SIZEOF(sL_BLK_SA[1]),         pBlockArray := ADR(sL_BLK_SA));
sMappingInfo.addBlkAry( iAdsBlockType := TO_UINT(ePr_BLK_SUBSTRATE),aAdsBlockName := 'sAdsSubstrate',       iAdsBlockVersion:= INT_TO_UINT(sAdsSubstrate[1].iO_Version),       iNbrBlocks := SIZEOF(sL_BLK_SUB)/SIZEOF(sL_BLK_SUB[1]),       pBlockArray := ADR(sL_BLK_SUB));
sMappingInfo.addBlkAry( iAdsBlockType := TO_UINT(ePr_BLK_CAMERA),   aAdsBlockName := 'sAdsCamera',          iAdsBlockVersion:= INT_TO_UINT(sAdsCamera[1].iO_Version),          iNbrBlocks := SIZEOF(sL_BLK_CAMERA)/SIZEOF(sL_BLK_CAMERA[1]), pBlockArray := ADR(sL_BLK_CAMERA));
sMappingInfo.bReady := TRUE;


(********************************* END OF ACTION *************************************************)
END_METHOD

METHOD RemVar
VAR
  lCtr : INT;
END_VAR
(*==== INIT ====*)
IF bL_InitRemVar THEN
  (*read remanet variables*)
  bL_InitRemVar := FALSE;

  (* -- Recipe read/write -------------------------------------------------------------------------*)
  IF pFbRecipeMngr = 0 THEN
    pFbRecipeMngr := PRG_SYSTEMBASE.fbRecipeAutoMngmt.register(
      aI_RecipePath           := CONCAT(aC_PlcConfigPath, aC_PlcRecipeSubPath),
      aI_RecipeDefinitionName := sC_Ads_Info.aType  (*is set in Mapping*)
    );
    FOR lCtr := 1 TO iCPr_NB_PM DO
      PRG_SYSTEMBASE.fbRecipeAutoMngmt.register(
        aI_RecipePath           := CONCAT(aC_PlcConfigPath, aC_PlcRecipeSubPath),
        aI_RecipeDefinitionName := F_Concat2('PRG_PRINT_PM', TO_STRING(lCtr))
      );
    END_FOR    
  END_IF

  (*load initial values if pattern was invalid*)
  IF sR_RemVar_P.aL_Pattern <> 16#ABCD THEN

    (*clear invalid persistence memory*)
    MEMSET(destAddr := ADR(sR_RemVar_P), 0, SIZEOF(ST_REM_VAR_P));
    
    (*initial boot values of project*)
    sR_RemVar_P.aL_Pattern := 16#ABCD;

    FOR lCtr := 1 TO iCPr_NB_PU DO

      sAdsSheetAlignment  [lCtr].bI_UsePrintMark         := TRUE;
      sAdsSheetAlignment  [lCtr].sI_PrintMarkSizeX.fI_Val:= 12.0; (*mm*)
      sAdsSheetAlignment  [lCtr].sI_PrintMarkSizeY.fI_Val:=  6.0; (*mm*)
      sAdsSheetAlignment  [lCtr].sI_HeadGap.fI_Val       :=  1.3; (*mm*)

//      Fb_PaperP_Detect_Cam[lCtr].iI_CurrentTimeStampComp := 2_000;
//      Fb_PaperP_Detect_Cam[lCtr].iI_SensorTimeStampComp  := 150;

    END_FOR;

    sAdsPrintGroup[ePr_PG_GROUP_1].sI_ShiftPositionX.lI_Val   := 100_000; (*um*)
    sAdsPrintGroup[ePr_PG_GROUP_2].sI_ShiftPositionX.lI_Val   := 200_000; (*um*)
    sAdsPrintGroup[ePr_PG_GROUP_3].sI_ShiftPositionX.lI_Val   := 300_000; (*um*)
    sAdsPrintGroup[ePr_PG_GROUP_4].sI_ShiftPositionX.lI_Val   := 400_000; (*um*)

    (*--- PC ---*)
    FOR lCtr := 1 TO iCPr_NB_PC DO
      sAdsPrintController[lCtr].sI_EnableHeater.bI_SetBool := TRUE;
      sAdsPrintController[lCtr].sI_EnablePrint .bI_SetBool := TRUE;
    END_FOR;

    (*--- PH ---*)
    FOR lCtr := 1 TO iCPr_NB_PH DO
      sAdsPrintHead[lCtr].aI_MaskFileName               := 'mask.msk';
      sAdsPrintHead[lCtr].aI_WaveFileName               := 'waveform.wav';
      sAdsPrintHead[lCtr].sI_VoltageScale.fI_Val        := 100;
    END_FOR;

    (*Recipe: write last recipe values*)
    IF pFbRecipeMngr <> 0 THEN
      pFbRecipeMngr^.mWriteRecipe(aSubName:='');
      PRG_MACHINE.bI_RecipeValuesLoadedPrint := TRUE;
    END_IF;

  ELSE

    (*--- PU ---*)
    FOR lCtr := 1 TO iCPr_NB_PU DO
      sAdsPrintUnit[lCtr].bI_Enable                     := sR_RemVar_P.bL_sAdsPrintUnit_bI_Enable[lCtr];

      sAdsPrintUnit[lCtr].sI_ShiftJobX.lI_Val           := sR_RemVar_P.lL_sAdsPrintUnit_sI_ShiftJobX[lCtr];
      sAdsPrintUnit[lCtr].sI_ShiftJobY.lI_Val           := sR_RemVar_P.lL_sAdsPrintUnit_sI_ShiftJobY[lCtr];

      sAdsSheetAlignment[lCtr].bI_UsePrintMark          := sR_RemVar_P.bL_WithMark;
      sAdsSheetAlignment[lCtr].sI_PrintMarkSizeX.fI_Val := sR_RemVar_P.fL_MarkLength;
      sAdsSheetAlignment[lCtr].sI_PrintMarkSizeY.fI_Val := sR_RemVar_P.fL_MarkHeigth;
    END_FOR;



    (*--- PG ---*)
    FOR lCtr := 1 TO iCPr_NB_PG DO
      sAdsPrintGroup [lCtr].bI_Enable                   := sR_RemVar_P.rL_sAdsPrintGroup_bI_Enable        [lCtr];
      sAdsPrintGroup [lCtr].sI_ShiftPositionX.lI_Val    := sR_RemVar_P.rL_sAdsPrintGroup_iO_PositionX     [lCtr];
      sAdsPrintGroup [lCtr].sI_ShiftPositionY.lI_Val    := sR_RemVar_P.rL_sAdsPrintGroup_iO_StartPositionX[lCtr];
    END_FOR;

    (*--- PC ---*)
    FOR lCtr := 1 TO iCPr_NB_PC DO
      sAdsPrintController[lCtr].bI_Enable                  := sR_RemVar_P.rL_sAdsPrintController      [lCtr];
      sAdsPrintController[lCtr].sI_EnableHeater.bI_SetBool := sR_RemVar_P.rL_sAdsPrintControllerHeater[lCtr];
      sAdsPrintController[lCtr].sI_EnablePrint .bI_SetBool := sR_RemVar_P.rL_sAdsPrintControllerPrint [lCtr];
    END_FOR;

    (*--- PH ---*)
    FOR lCtr := 1 TO iCPr_NB_PH DO
      sAdsPrintHead[lCtr].bI_Enable                     := sR_RemVar_P.rL_sAdsPrintHead_bI_Enable        [lCtr];
      sAdsPrintHead[lCtr].sI_ShiftPositionX.lI_Val      := sR_RemVar_P.rL_sAdsPrintHead_iO_PositionX     [lCtr];
      sAdsPrintHead[lCtr].sI_PositionX.lI_Val           := sR_RemVar_P.rL_sAdsPrintHead_iO_StartPositionX[lCtr];
      sAdsPrintHead[lCtr].sI_PositionY.lI_Val           := sR_RemVar_P.rL_sAdsPrintHead_iO_StartPositionY[lCtr];
      sAdsPrintHead[lCtr].aI_MaskFileName               := sR_RemVar_P.rL_sAdsPrintHead_aI_MaskFileName  [lCtr];
      sAdsPrintHead[lCtr].aI_WaveFileName               := sR_RemVar_P.rL_sAdsPrintHead_aI_WaveFileName  [lCtr];
      sAdsPrintHead[lCtr].sI_VoltageScale.fI_Val        := sR_RemVar_P.rL_sAdsPrintHead_fI_VoltScale     [lCtr];
    END_FOR;

  END_IF;

(*************************************************************************************************)
(********************************* WRITING REMANENT VARIABLES ************************************)
(*************************************************************************************************)
ELSE
  (* ------ Update Remanent values --------- *)

  (*--- PU ---*)
  FOR lCtr:=1 TO iCPr_NB_PU DO
    sR_RemVar_P.bL_sAdsPrintUnit_bI_Enable[lCtr]          := sAdsPrintUnit[lCtr].bI_Enable;

    sR_RemVar_P.lL_sAdsPrintUnit_sI_ShiftJobX[lCtr]       := sAdsPrintUnit[lCtr].sI_ShiftJobX.lI_Val;
    sR_RemVar_P.lL_sAdsPrintUnit_sI_ShiftJobY[lCtr]       := sAdsPrintUnit[lCtr].sI_ShiftJobY.lI_Val;


    sR_RemVar_P.bL_WithMark                               := sAdsSheetAlignment[lCtr].bI_UsePrintMark;
    sR_RemVar_P.fL_MarkLength                             := sAdsSheetAlignment[lCtr].sI_PrintMarkSizeX.fI_Val;
    sR_RemVar_P.fL_MarkHeigth                             := sAdsSheetAlignment[lCtr].sI_PrintMarkSizeY.fI_Val;

  END_FOR;

  (*--- PG ---*)
  FOR lCtr:=1 TO iCPr_NB_PG DO
    sR_RemVar_P.rL_sAdsPrintGroup_bI_Enable        [lCtr] := sAdsPrintGroup [lCtr].bI_Enable;
    sR_RemVar_P.rL_sAdsPrintGroup_iO_PositionX     [lCtr] := sAdsPrintGroup [lCtr].sI_ShiftPositionX.lI_Val;
    sR_RemVar_P.rL_sAdsPrintGroup_iO_StartPositionX[lCtr] := sAdsPrintGroup [lCtr].sI_ShiftPositionY.lI_Val;
  END_FOR;

  (*--- PC ---*)
  FOR lCtr:=1 TO iCPr_NB_PC DO
    sR_RemVar_P.rL_sAdsPrintController             [lCtr] := sAdsPrintController[lCtr].bI_Enable;
    sR_RemVar_P.rL_sAdsPrintControllerHeater       [lCtr] := sAdsPrintController[lCtr].sI_EnableHeater.bI_SetBool;
    sR_RemVar_P.rL_sAdsPrintControllerPrint        [lCtr] := sAdsPrintController[lCtr].sI_EnablePrint .bI_SetBool;
  END_FOR;

  (*--- PH ---*)
  FOR lCtr:=1 TO iCPr_NB_PH DO
    sR_RemVar_P.rL_sAdsPrintHead_bI_Enable         [lCtr] := sAdsPrintHead[lCtr].bI_Enable;
    sR_RemVar_P.rL_sAdsPrintHead_iO_PositionX      [lCtr] := sAdsPrintHead[lCtr].sI_ShiftPositionX.lI_Val;
    sR_RemVar_P.rL_sAdsPrintHead_iO_StartPositionX [lCtr] := sAdsPrintHead[lCtr].sI_PositionX.lI_Val;
    sR_RemVar_P.rL_sAdsPrintHead_iO_StartPositionY [lCtr] := sAdsPrintHead[lCtr].sI_PositionY.lI_Val;
    sR_RemVar_P.rL_sAdsPrintHead_aI_MaskFileName   [lCtr] := sAdsPrintHead[lCtr].aI_MaskFileName;
    sR_RemVar_P.rL_sAdsPrintHead_aI_WaveFileName   [lCtr] := sAdsPrintHead[lCtr].aI_WaveFileName;
    sR_RemVar_P.rL_sAdsPrintHead_fI_VoltScale      [lCtr] := sAdsPrintHead[lCtr].sI_VoltageScale.fI_Val;
  END_FOR;

END_IF;
END_METHOD

METHOD PRIVATE setLoggingLevels
VAR_INPUT
END_VAR
(*Configure logging*)
LogPrSetup.LogLevel                  := ePrint_LogLevel;
FB_PU[ePr_PU_UNIT_1].LogLevel        := ePrint_LogLevel;
fbPm.LogLevel                        := ePrint_LogLevel;
fbModuleMaster.LogLevel              := ePrint_LogLevel;
END_METHOD

METHOD PRIVATE setupAdsPc
VAR_INPUT
  pAds : POINTER TO ST_ADS_PC;
  nIdx : UDINT;
END_VAR
pAds^.aO_Name 							        := sC_Config_P.aC_PC_NAME[nIdx];
//pAds^.bI_Enable                     := TRUE;   // use persistence
pAds^.bO_EnableExist                := TRUE;
pAds^.sI_EnableHeater.bC_BoolExist  := TRUE;
pAds^.sI_EnableHeater.bO_BoolCanSet := TRUE;
pAds^.sI_EnablePrint .bC_BoolExist  := TRUE;
pAds^.sI_EnablePrint .bO_BoolCanSet := TRUE;
END_METHOD

METHOD PRIVATE setupAdsPg
VAR_INPUT
  pAds : POINTER TO ST_ADS_PG;
  nIdx : UDINT;
END_VAR
pAds^.aO_Name:=sC_Config_P.aC_PG_NAME[nIdx];
pAds^.sI_ShiftPositionX.bC_Exist:=TRUE;
pAds^.sI_ShiftPositionX.aC_Unit:=sC_Config_P.aC_xx_STARTPOS_X_UNIT;
pAds^.sI_ShiftPositionX.lC_Min:=sC_Config_P.lL_xx_STARTPOS_X_SET_MIN;
pAds^.sI_ShiftPositionX.lC_Max:=sC_Config_P.lL_xx_STARTPOS_X_SET_MAX;
pAds^.sI_ShiftPositionY.bC_Exist:=FALSE;
pAds^.sI_ShiftPositionY.aC_Unit:=sC_Config_P.aC_xx_STARTPOS_Y_UNIT;
pAds^.sI_ShiftPositionY.lC_Min:=sC_Config_P.lL_xx_STARTPOS_Y_SET_MIN;
pAds^.sI_ShiftPositionY.lC_Max:=sC_Config_P.lL_xx_STARTPOS_Y_SET_MAX;
pAds^.sI_CommandChangeInk.bO_CommandExist:=FALSE;
pAds^.sI_CommandChangeInk.bO_CommandCanEx:=FALSE;
pAds^.sI_CommandEmptyInk.bO_CommandExist:=FALSE;
pAds^.sI_CommandEmptyInk.bO_CommandCanEx:=FALSE;
END_METHOD

METHOD PRIVATE setupAdsPh
VAR_INPUT
  pAds : POINTER TO ST_ADS_PH;
  nIdx : UDINT;
END_VAR
pAds^.aO_Name 										:= sC_Config_P.aC_PH_NAME[nIdx];
pAds^.sI_PositionX.bC_Exist       := TRUE;
pAds^.sI_PositionX.aC_Type        := sC_Config_P.aC_xx_POSITION_X_TYPE;
pAds^.sI_PositionX.aC_Unit        := sC_Config_P.aC_xx_POSITION_X_UNIT;
pAds^.sI_PositionX.lC_Min         := sC_Config_P.lL_xx_POSITION_X_SET_MIN;
pAds^.sI_PositionX.lC_Max         := sC_Config_P.lL_xx_POSITION_X_SET_MAX;
pAds^.sI_PositionY.bC_Exist       := TRUE;
pAds^.sI_PositionY.aC_Type        := sC_Config_P.aC_xx_POSITION_X_TYPE;
pAds^.sI_PositionY.aC_Unit        := sC_Config_P.aC_PH_OFFSETPOS_Y_UNIT;
pAds^.sI_PositionY.lC_Min         := sC_Config_P.lL_PH_OFFSETPOS_Y_SET_MIN;
pAds^.sI_PositionY.lC_Max         := sC_Config_P.lL_PH_OFFSETPOS_Y_SET_MAX;
pAds^.sI_ShiftPositionX.bC_Exist  := FALSE;
pAds^.sI_ShiftPositionX.lC_Min    := sC_Config_P.lL_xx_POSITION_X_SET_MIN;
pAds^.sI_ShiftPositionX.lC_Max    := sC_Config_P.lL_xx_POSITION_X_SET_MAX;
pAds^.sI_ShiftPositionY.bC_Exist  := FALSE;
pAds^.sI_ShiftPositionY.lC_Min    := sC_Config_P.lL_PH_OFFSETPOS_Y_SET_MIN;
pAds^.sI_ShiftPositionY.lC_Max    := sC_Config_P.lL_PH_OFFSETPOS_Y_SET_MAX;
pAds^.sI_VoltageScale.bC_Exist    := TRUE;
pAds^.sI_VoltageScale.aC_Unit     := '%';
pAds^.sI_VoltageScale.fC_Min      := 90;
pAds^.sI_VoltageScale.fC_Max      := 110;
pAds^.cO_HeadIndex                := cCPr_MAP_PH_PC_INDEX[nIdx];
END_METHOD

METHOD PRIVATE setupAdsPm
VAR_INPUT
  pAds : POINTER TO ST_ADS_PM;
  nIdx : UDINT;
END_VAR
pAds^.aO_Name                     := sC_Config_P.aC_PM_NAME[nIdx];
pAds^.bI_Enable                   := TRUE;
pAds^.sI_GeneralShiftX.bC_Exist   := TRUE;
pAds^.sI_GeneralShiftX.aC_Unit    := sC_Config_P.aC_PU_GENERALSHIFT_X_UNIT;
pAds^.sI_GeneralShiftX.lC_Min     := sC_Config_P.lL_PU_GENERALSHIFT_X_SET_MIN;
pAds^.sI_GeneralShiftX.lC_Max     := sC_Config_P.lL_PU_GENERALSHIFT_X_SET_MAX;
pAds^.sI_GeneralShiftY.bC_Exist   := TRUE;
pAds^.sI_GeneralShiftY.aC_Unit    := sC_Config_P.aC_PU_GENERALSHIFT_Y_UNIT;
pAds^.sI_GeneralShiftY.lC_Min     := sC_Config_P.lL_PU_GENERALSHIFT_Y_SET_MIN;
pAds^.sI_GeneralShiftY.lC_Max     := sC_Config_P.lL_PU_GENERALSHIFT_Y_SET_MAX;
END_METHOD

METHOD PRIVATE setupAdsPu
VAR_INPUT
  pAds : POINTER TO ST_ADS_PU;
  nIdx : UDINT;
END_VAR
pAds^.aO_Name 										     := sC_Config_P.aC_PU_NAME[nIdx];
pAds^.sI_ShiftJobX.bC_Exist            := FALSE;
pAds^.sI_ShiftJobX.aC_Unit             := sC_Config_P.aC_PU_SHIFTPOS_X_UNIT;
pAds^.sI_ShiftJobX.lC_Min              := sC_Config_P.lL_PU_SHIFTPOS_X_SET_MIN;
pAds^.sI_ShiftJobX.lC_Max              := sC_Config_P.lL_PU_SHIFTPOS_X_SET_MAX;
pAds^.sI_ShiftJobY.bC_Exist            := FALSE;
pAds^.sI_ShiftJobY.aC_Unit             := sC_Config_P.aC_PU_SHIFTPOS_Y_UNIT;
pAds^.sI_ShiftJobY.lC_Min              := sC_Config_P.lL_PU_SHIFTPOS_Y_SET_MIN;
pAds^.sI_ShiftJobY.lC_Max              := sC_Config_P.lL_PU_SHIFTPOS_Y_SET_MAX;
pAds^.sO_StopRequestEvent.bC_Enable    := TRUE;
pAds^.sO_StopRequestEvent.bC_Exist     := TRUE;
pAds^.sO_StopRequestEvent.iC_CycleTime := 50;
END_METHOD

METHOD PRIVATE setupAdsSa
VAR_INPUT
  pAds : POINTER TO ST_ADS_DVTSHEETALIGNMENT;
END_VAR
pAds^.aO_Name                    := sC_Config_P.aC_SHEETALIGNMENT_NAME;
pAds^.sI_PrintMarkSizeX.bC_Exist := TRUE;
pAds^.sI_PrintMarkSizeX.aC_Unit  := sC_Config_P.aC_xx_PRINTMARK_X_UNIT;
pAds^.sI_PrintMarkSizeX.fC_Min   := sC_Config_P.fL_xx_PRINTMARK_X_SET_MIN;
pAds^.sI_PrintMarkSizeX.fC_Max   := sC_Config_P.fL_xx_PRINTMARK_X_SET_MAX;
pAds^.sI_PrintMarkSizeY.bC_Exist := TRUE;
pAds^.sI_PrintMarkSizeY.aC_Unit  := sC_Config_P.aC_xx_PRINTMARK_Y_UNIT;
pAds^.sI_PrintMarkSizeY.fC_Min   := sC_Config_P.fL_xx_PRINTMARK_Y_SET_MIN;
pAds^.sI_PrintMarkSizeY.fC_Max   := sC_Config_P.fL_xx_PRINTMARK_Y_SET_MAX;
pAds^.sI_HeadGap.bC_Exist        := TRUE;
pAds^.sI_HeadGap.aC_Unit         := sC_Config_P.aC_xx_HEAD_GAP_UNIT;
pAds^.sI_HeadGap.fC_Min          := sC_Config_P.fL_xx_HEAD_GAP_SET_MIN;
pAds^.sI_HeadGap.fC_Max          := sC_Config_P.fL_xx_HEAD_GAP_SET_MAX;
pAds^.sO_CurrentAngle.bC_Exist   := FALSE;
pAds^.sO_CurrentAngle.aC_Unit    := sC_Config_P.aC_xx_CURRENT_ANGLE_UNIT;
pAds^.sO_CurrentAngle.fC_Min     := sC_Config_P.fL_xx_CURRENT_ANGLE_SET_MIN;
pAds^.sO_CurrentAngle.fC_Max     := sC_Config_P.fL_xx_CURRENT_ANGLE_SET_MAX;
END_METHOD

METHOD PRIVATE setupAdsSub
VAR_INPUT
  pAds : POINTER TO ST_ADS_SUBSTRATE;
  nIdx : UDINT;
END_VAR
pAds^.aO_Name                     := CONCAT(sC_Config_P.aC_SUB_NAME, TO_STRING(nIdx));
pAds^.sI_SurfaceVelocity.bC_Exist := FALSE;
pAds^.sI_SurfaceVelocity.aC_Type  := sC_Config_P.aC_SUB_SURFACE_VELOCITY_TYPE;
pAds^.sI_SurfaceVelocity.aC_Unit  := sC_Config_P.aC_SUB_SURFACE_VELOCITY_UNIT;
pAds^.sI_SurfaceVelocity.fC_Min   := sC_Config_P.fC_SUB_SURFACE_VELOCITY_SET_MIN;
pAds^.sI_SurfaceVelocity.fC_Max   := sC_Config_P.fC_SUB_SURFACE_VELOCITY_SET_MAX;
pAds^.sI_SizeX.bC_Exist           := FALSE;
pAds^.sI_SizeX.aC_Unit            := sC_Config_P.aC_SUB_SURFACE_SIZE_UNIT;
pAds^.sI_SizeX.fC_Min             := sC_Config_P.fC_SUB_SURFACE_SIZE_SET_MIN;
pAds^.sI_SizeX.fC_Max             := sC_Config_P.fC_SUB_SURFACE_SIZE_SET_MAX;
pAds^.sI_SizeY.bC_Exist           := FALSE;
pAds^.sI_SizeY.aC_Unit            := sC_Config_P.aC_SUB_SURFACE_SIZE_UNIT;
pAds^.sI_SizeY.fC_Min             := sC_Config_P.fC_SUB_SURFACE_SIZE_SET_MIN;
pAds^.sI_SizeY.fC_Max             := sC_Config_P.fC_SUB_SURFACE_SIZE_SET_MAX;
pAds^.sI_SizeZ.bC_Exist           := FALSE;
pAds^.sI_SizeZ.aC_Unit            := sC_Config_P.aC_SUB_SURFACE_SIZE_UNIT;
pAds^.sI_SizeZ.fC_Min             := sC_Config_P.fC_SUB_SURFACE_SIZE_SET_MIN;
pAds^.sI_SizeZ.fC_Max             := sC_Config_P.fC_SUB_SURFACE_SIZE_SET_MAX;
pAds^.sI_PositionX.bC_Exist       := FALSE;
pAds^.sI_PositionX.aC_Unit        := sC_Config_P.aC_SUB_SURFACE_POS_UNIT;
pAds^.sI_PositionX.fC_Min         := sC_Config_P.fC_SUB_SURFACE_POS_SET_MIN;
pAds^.sI_PositionX.fC_Max         := sC_Config_P.fC_SUB_SURFACE_POS_SET_MAX;
pAds^.sI_PositionY.bC_Exist       := FALSE;
pAds^.sI_PositionY.aC_Unit        := sC_Config_P.aC_SUB_SURFACE_POS_UNIT;
pAds^.sI_PositionY.fC_Min         := sC_Config_P.fC_SUB_SURFACE_POS_SET_MIN;
pAds^.sI_PositionY.fC_Max         := sC_Config_P.fC_SUB_SURFACE_POS_SET_MAX;
pAds^.sI_PositionZ.bC_Exist       := FALSE;
pAds^.sI_PositionZ.aC_Unit        := sC_Config_P.aC_SUB_SURFACE_POS_UNIT;
pAds^.sI_PositionZ.fC_Min         := sC_Config_P.fC_SUB_SURFACE_POS_SET_MIN;
pAds^.sI_PositionZ.fC_Max         := sC_Config_P.fC_SUB_SURFACE_POS_SET_MAX;
END_METHOD

METHOD Testing : BOOL
VAR_INPUT
END_VAR
VAR
  nCt, nRun : DINT;
  eLogLevel : E_LogSeverity;
END_VAR
//-------------------------------------------------------------
// Test handler for PRG_PRINT specific tasks. 
// Here we have full access to all PRG_PRINT internal elements.
//-------------------------------------------------------------

//-------------------------------------------------------
PRG_TEST();     // call the other PRG_TEST code
//-------------------------------------------------------

//-------------------------------------------------------
// test tasks 

//- testing disabled completely  
IF NOT fbPrgPrintTest.bEnTesting THEN 
  RETURN;
END_IF

//- Initialize the testing at start  
IF NOT fbPrgPrintTest.bInitialized THEN 
  fbPrgPrintTest.Init(
    pAdsPu:=ADR(sAdsPrintUnit[1]), 
    pAdsCamera:=ADR(sAdsCamera[1]),
    pAdsSubstrate:=ADR(sAdsSubstrate[1])
  ); 
  RETURN;
END_IF

//- Enter machine into testing mode
IF fbPrgPrintTest.bEnterSim THEN
    LogPrSetup.LogWarning('Start print testing...');
    // configure persistences (if they were lost)
    sAdsPrintGroup[1].bI_Enable := TRUE;
    sAdsPrintGroup[2].bI_Enable := FALSE;
    sAdsPrintController[1].bI_Enable := TRUE;
    sAdsPrintController[1].sI_EnableHeater.bI_SetBool := TRUE;
    sAdsPrintController[1].sI_EnablePrint.bI_SetBool := TRUE;
    sAdsPrintHead[1].iI_Temperature := 500;
    // global worker
    fbWorkerVerify.bWorkerEnable := TRUE;
    fbWorkerDelete.bWorkerEnable := TRUE;
END_IF
//- Exit machine from testing mode (may need a restart completely, values before test were not persisted)
IF fbPrgPrintTest.bExitSim THEN
    LogPrSetup.LogWarning('Stop print testing...');   
    // exit simulation mode
    //fbPrintModule[1].bSimEnable := FALSE;
END_IF
IF fbPrgPrintTest.bStartMachine THEN
    LogPrSetup.LogWarning('Start machine...');
    fbPrgPrintTest.bSimPrgMachine := TRUE;
    fbPrintModule[1].bSimEnable := TRUE;
END_IF
IF fbPrgPrintTest.bStopMachine THEN
    LogPrSetup.LogWarning('Stop machine...');
    fbPrgPrintTest.bSimPrgMachine := FALSE;
    fbPrintModule[1].bSimEnable := FALSE;
END_IF
//- log level management
IF fbPrgPrintTest.isLogLevelUpdate(eLogSeverity=>eLogLevel) THEN
    // TODO: implement something similar in PrintModule simaulation
    PRG_PRINT.fbWorkerVerify.LogLevel := eLogLevel;
    PRG_PRINT.fbWorkerDelete.LogLevel := eLogLevel;
    PRG_PRINT.LogPrSetup.LogLevel := eLogLevel;
END_IF

fbPrgPrintTest(); // call test fb

// distribute simulation mode to PRGs
IF fbPrgPrintTest.bChangedPrgSim THEN
  PRG_PRINT.bSimulation := fbPrgPrintTest.bSimPrgPrint;
  PRG_MACHINE.bSimulation := fbPrgPrintTest.bSimPrgMachine;
  PRG_INK.bSimulation := fbPrgPrintTest.bSimPrgInk;
END_IF
END_METHOD

END_PROGRAM

// ---- POUs/Products/Print_Weu/FB_PrintModule_WEU.TcPOU
FUNCTION_BLOCK FB_PrintModule_WEU EXTENDS FB_PrintModule_Base
VAR_INPUT
  fPUPlate1_Temperature : LREAL;  // PU Plate1 temperature
  fPUPlate2_Temperature : LREAL;  // PU Plate2 temperature
END_VAR
VAR
  (* Module specific sub-modules - WEU module contains a 
    - print position (encoder input to print domain translation)
    - Mark sensor with a mark detection module which provices a camera trigger and start position detection
    - Mark definition (used by the detection and camera)
  *)
  fbPrintPosition    : FB_PrintPositionDmax;   // a position per pm (external encoder wheel)
  fbMarkDefinition   : FB_MarkDefinition;      // mark definition instance (used by MarkDetection and camera)
  fbMarkDetection    : FB_MarkDetection;       // StartPosTrigger, CameraTrigger and MarkDetection (Mark handler for MarkCamera)
  fbMarkCameraWeu    : FB_MarkCamera_WEU;      // Mark detection camera
  fbNoCamera         : FB_CameraDummy;         // dummy sheet detect camera (not actively used)
  
  // additional grid corrections
  // - PU Deformation/correction (4p, banana, ...)
  fbFineAlignement   : FB_FineAlignement;
  // view
  fbView             : FB_PrintModule_WEU_View;    // additional controls for print module visus
END_VAR
VAR PERSISTENT
  _fEncoderCylinderDiameter : LREAL := 100.0;      // Encoder cylinder diameter [mm]
END_VAR
VAR CONSTANT
  fC_EncoderImpU : LREAL := 10_000 * 4;   // Impulses * 4 times sampling [Imp/U]
END_VAR

IF NOT bInit THEN RETURN; END_IF

// - calculate encoder resolution (fL_SubstrateThickness with factor is added to the radius because of the neutral fiber of the substrate)
//   update encoder position based on machine parameter
_iPrintPosition.fEnoderResolution := ((_fEncoderCylinderDiameter / 1000 / 2) + (_pModuleMachineState^.fSubstrateThickness * (_pModuleMachineState^.fNeutralFibreFactor) / 100)) * 2 * PI * 1_000_000 / fC_EncoderImpU;
fbPrintPosition();

//fbMarkDefinition();   // no call to body 
fbMarkDetection(
  bEnable:=bReadyForPrinting,
  bAutomaticMode:=TRUE,
  nCurrentPos:=_iPrintPosition.getPosition(),
  fCurrentSpeed:=_iPrintPosition.getSpeed()
);

fbMarkCameraWeu();
fbNoCamera();

(*PU corrections*)
IF GVL_Deformation.bC_UsePUDeformation THEN
  fbFineAlignement.fT_PL1 := fPUPlate1_Temperature;
  fbFineAlignement.fT_PL2 := fPUPlate2_Temperature;
  fbFineAlignement();
END_IF

fbView();

// call module base
SUPER^();

// simulation
SimUpdate();

// machine interface outputs
_pModuleMachineFeedback^.nPrintMarkPosBits := fbMarkDetection.nPrintMarkPosBits;

METHOD Init : BOOL
VAR_INPUT
  nIdx                  : UDINT;                                // Module id
  pAdsPm                : POINTER TO ST_ADS_PM;                 // ADS module
  pAdsSa                : POINTER TO ST_ADS_DVTSHEETALIGNMENT;  // ADS sheet alignement
  pAdsCam               : POINTER TO ST_ADS_CAMERA;             // ADS camera
  pAdsPg                : ARRAY[1..GVL_WEU.nC_WorkerPrintPerPm] OF POINTER TO ST_ADS_PG;  // PG -> worker ads 
  
  // config print
  fCycleTime            : LREAL;                // task cycle time in [s]
  fPrintUnitWidth       : LREAL;                // PrintUnit width mechanical [m]
  nYShiftPcCenter       : UDINT;                // Y shift for centered image data in RAM [px]
  // references
  iModuleMaster         : I_ModuleMaster;       // interface for module to master (main) communication
  iPosition             : I_PrintPosition;      // interface for print position
  iStartPos             : I_StartPosDetect;     // interface for start position detect
  iSystemStatus         : I_SystemStatus;       // system status interface (for sleep, estop, ...), may shadow states from machine inputs
  pMachineInputs        : POINTER TO ST_ModuleMachineInterface_IN;
  pMachineOutputs       : POINTER TO ST_ModuleMachineInterface_OUT;
END_VAR
VAR
  nCtr : UDINT;
END_VAR
IF iPosition = 0 THEN _iPrintPosition := fbPrintPosition;     // select internal print position if not given externally
ELSE                  _iPrintPosition := iPosition; END_IF

fbPrintPosition.Init(fPrintResolution:=_iPrintPosition.fPrintResolution, fSubPxResolution:=_iPrintPosition.fSubPxResolution, fTaskCycleTime:=fCycleTime);
// -- Mark definition handler
fbMarkDefinition.Init();
// -- Sheet/Camera trigger & mark detection
fbMarkDetection.Init(fPrintResolution:=_iPrintPosition.fPrintResolution, fSubPxResolution:=_iPrintPosition.fSubPxResolution, pFbMarkDefinition:=ADR(fbMarkDefinition));

// -- Mark camera
fbMarkCameraWeu.InitMarkCamera(nPrintUnitResolution:=TO_UDINT(_iPrintPosition.fPrintResolution), nPrintUnitSubPx:=TO_UDINT(_iPrintPosition.fSubPxResolution), iCameraTrigger:=fbMarkDetection, iMarkDefinition:=fbMarkDefinition);
fbMarkCameraWeu.sVisuName := 'VISU_MarkCamera_WEU';
fbWorkerCamera.RegisterCamera(fbMarkCameraWeu);

// -- Camera if mark is not selected
fbNoCamera.Init(nPrintUnitResolution:=TO_UDINT(_iPrintPosition.fPrintResolution), nPrintUnitSubPx:=TO_UDINT(_iPrintPosition.fSubPxResolution), iCameraTrigger:=fbMarkDetection, bUseCameraTrigger:=FALSE, bUseCameraTriggerFeedback:=FALSE);
fbWorkerCamera.RegisterCamera(fbNoCamera);


SUPER^.Init(
  nIdx              := nIdx,
  pAdsPm            := pAdsPm,
  pAdsSa            := pAdsSa,
  pAdsCam           := pAdsCam,
  pAdsPg            := pAdsPg,
  // config print
  fCycleTime        := fCycleTime,
  fPrintUnitWidth   := fPrintUnitWidth,
  nYShiftPcCenter   := nYShiftPcCenter,
  // references     
  iModuleMaster     := iModuleMaster,     // internal subm
  iPosition         := fbPrintPosition,   // internal subm
  iStartPos         := fbMarkDetection,   // internal subm
  iSystemStatus     := iSystemStatus, 
  pMachineInputs    := pMachineInputs,
  pMachineOutputs   := pMachineOutputs
);

// additional grid point corrections
fbFineAlignement.init(pAdsCam := pAdsCam, fPxReso := _iPrintPosition.fPrintResolution, fPuWidth := fPrintUnitWidth);
// - register them to workers
FOR nCtr := 1 TO GVL_WEU.nC_WorkerPrintPerPm DO
  fbWorkerPrint[nCtr].RegisterGridCorrection(iGridCorrection:=fbFineAlignement);
END_FOR 

fbView.init(pModule:=THIS, pPositioning:=ADR(fbPrintPosition));
setLogLevels(lvl:=E_LogSeverity.Debug);
END_METHOD

METHOD PROTECTED setLogLevels
VAR_INPUT
  lvl : E_LogSeverity;
END_VAR
// - base
SUPER^.setLogLevels(lvl:=lvl);
// - weu
fbPrintPosition.LogLevel := lvl;
fbMarkDefinition.LogLevel := lvl;
fbMarkDetection.LogLevel := lvl;
fbMarkCameraWeu.LogLevel := lvl;
fbNoCamera.LogLevel := lvl;
END_METHOD

METHOD PRIVATE SimUpdate
VAR_INPUT
END_VAR
VAR_INST
  rfTrig_SimEnable : RF_TRIG;
END_VAR
rfTrig_SimEnable(CLK:=_bSimEnable);
IF    rfTrig_SimEnable.RT THEN
  // ev. enable
  //fbWorkerCamera.bWorkerEnable := TRUE;
  //fbWorkerDeformation.bWorkerEnable := TRUE;
  //fbWorkerPrint[1].bWorkerEnable := TRUE;
  //fbWorkerPrint[2].bWorkerEnable := TRUE;
  
  fbPrintPosition.bSimEnable  := TRUE;
  //fbMarkDefinition
  fbMarkDetection.bSimEnable := TRUE;
  fbMarkCameraWeu.bSimulate := TRUE;

ELSIF rfTrig_SimEnable.FT THEN
  // ev. disable
  fbPrintPosition.bSimEnable  := FALSE;
  fbMarkDetection.bSimEnable := FALSE;
  fbMarkCameraWeu.bSimulate := FALSE;

ELSIF _bSimEnable THEN
  // enabled
  ;
ELSE
  ; // disabled
END_IF
END_METHOD

END_FUNCTION_BLOCK

// ---- POUs/Products/Print_Weu/FB_PrintModule_Base.TcPOU
(*
  A DVT PrintModule (DEU, DSU, WEU).
*)
FUNCTION_BLOCK FB_PrintModule_Base EXTENDS FB_Sim
VAR_INPUT
  // encoder input --> directly mapped into FB_PrintPosition 
  // machine state by pointer in init()
  // external start pos interface by pointer in init()
  fPrintOffsetX  : ARRAY[1..GVL_WEU.nC_WorkerPrintPerPm] OF LREAL;   // external configurative offsets to PM (PU / PM /PG) 
  fPrintOffsetY  : ARRAY[1..GVL_WEU.nC_WorkerPrintPerPm] OF LREAL;   // external configurative offsets to PM (PU / PM / PG / Machine) 
END_VAR

VAR
  //config
  _nIdx                   : UDINT;        // for visu selection only (remove later)
  _pAdsPm                 : POINTER TO ST_ADS_PM; //ads config/status interface
  _pAdsSa                 : POINTER TO ST_ADS_DVTSHEETALIGNMENT; // sheet alignemnt ads
  
  _nYShift_PcRamCenter    : UDINT;        // y-shift for centered image in CB RAM [px]
  
  // - references
  _iModuleMaster          : I_ModuleMaster;       // master module (setting, position, global stuff, ...)
  _iPrintPosition         : I_PrintPosition;      // module's position
  _iStartPos              : I_StartPosDetect;     // module's start position detect
  _iSystemStatus          : I_SystemStatus;       // module's system status
  _pModuleMachineState    : POINTER TO ST_ModuleMachineInterface_IN;   // machine interface-print states
  _pModuleMachineFeedback : POINTER TO ST_ModuleMachineInterface_OUT;  // machine interface-print feedback
    
  // status
  bInit                   : BOOL;   // initialized
  bReadyForPrinting       : BOOL;   // Module ready for printing
  bHardwareHold           : BOOL;   // hw hold
  
  // instances
  fbParamMediator         : FB_DefGridParamMediator;
  fbWorkerCamera          : FB_WorkerDefGrid_Camera;
  fbWorkerPrint           : ARRAY[1..GVL_WEU.nC_WorkerPrintPerPm] OF FB_WorkerDefGrid_Print_WEU;
  fbWorkerDeformation     : FB_WorkerDefGrid_Deformation;
  
  // hw (references only for now) ------
  // - pc
  _pPc                    : ARRAY[1..GVL_WEU.nC_MaxPcPerPm] OF POINTER TO FB_PC;
  _nPc                    : UDINT;  // number of PC in module
  _nPcToWorker_Mapping    : ARRAY[1..GVL_WEU.nC_MaxPcPerPm] OF UDINT;  // Mapping of PC to worker
  // - ph
  _pPh                    : ARRAY[1..GVL_WEU.nC_MaxPhPerPm] OF POINTER TO FB_PH_Grid;
  _nPh                    : UDINT;  // number of PH in module
  _nPhToWorker_Mapping    : ARRAY[1..GVL_WEU.nC_MaxPhPerPm] OF UDINT;  // Mapping of PH to worker
  _nPhToPc_Mapping        : ARRAY[1..GVL_WEU.nC_MaxPhPerPm] OF UDINT;  // Mapping of PH to PC
  _nPhToPcCh_Mapping      : ARRAY[1..GVL_WEU.nC_MaxPhPerPm] OF UDINT;  // Mapping of PH to PC channel
  
  // helper
  nCtr                    : UDINT;
  fSpeed, fSpeedMpMin     : LREAL;
  bProductionSpeedReached : BOOL;
  fPuElevation            : LREAL;
  nPos_SubPx, nPos_Px     : DINT;
  nPos_SubPx_mem          : DINT;
  fPos_um                 : LREAL;
  rT_SyncRequest          : R_TRIG;
  tSyncDelay              : TON;
  bHwSyncCmd              : BOOL;
 
  // messaging
  fb_MsgQueue             : FB_MSG_QUEUE;                 (*Message queue*)
  fb_MsgHandler           : FB_MSG_HANDLER;               (*Message handler*)
  sL_MsgConfig            : ST_MSG_CONFIG;                (*Message config*)
  fb_Msg                  : ARRAY [1..nC_NumMsg] OF FB_MESSAGE;  (*Messages*)
  
END_VAR
VAR PERSISTENT
  _fDistToMasterPm        : LREAL;  // distance to master reference module (mech.), does not include DetectToPu
  _fPrintModuleAdjustY    : LREAL;  // Module adjust Y [µm]*)
END_VAR
VAR CONSTANT
  fC_HeadOffsetPlate      : LREAL := 0.000_2;      // Head offset to base plate [m]
  fC_ProductionSpeedMpMin_Level   : LREAL := 5.0;          // [m/min]
  nC_NumMsg               : INT := 8;              // number of internal messages
END_VAR

IF NOT bInit THEN RETURN; END_IF
SUPER^();

bReadyForPrinting :=    _pModuleMachineState^.bEngaged 
                     AND _pModuleMachineState^.bPrintEnabled 
                     AND _pModuleMachineState^.bUnitInPrintPosition
                     AND NOT _pModuleMachineState^.bEStop
                     AND NOT _pModuleMachineState^.bSleep;

// sync trigger generation
rT_SyncRequest(CLK:=bReadyForPrinting);
IF rT_SyncRequest.Q THEN  // OR rT_JobActive.Q 
  tSyncDelay(IN:=TRUE, PT:=T#2MS);   // a Sync delay to workaround a sync sent to CB while a Start or Prepare Command
END_IF
tSyncDelay(Q=>bHwSyncCmd); 
IF tSyncDelay.Q THEN 
  tSyncDelay(IN:=FALSE);
END_IF

// positioning
fSpeed     := _iPrintPosition.getSpeed(fSpeedMpMin=>fSpeedMpMin);
bProductionSpeedReached := (fSpeedMpMin >= fC_ProductionSpeedMpMin_Level);
// get position (hide encoder if not ready for printing or moving)
nPos_SubPx := _iPrintPosition.getPosition(nPosition_px=>nPos_Px, fPosition_um=>fPos_um);

// security measures (jetting when not really moving or not in position)
nPos_SubPx := nPos_SubPx_mem := SEL(bReadyForPrinting AND _iPrintPosition.bMoving, nPos_SubPx_mem, nPos_SubPx);
// what happens when PM slows down e.g. notaus with endless printing (safety measure), maybe not needed with new Jm (stop after a repeat)
 // - enabled & > minimum speed
 // - enabled & > production min speed
bHardwareHold := NOT bProductionSpeedReached OR NOT _pModuleMachineState^.bPrintEnabled;  // Hw HOLD: 
{warning '@HOA TODO what value is this, from where'}
fPuElevation := LIMIT(0, (_pAdsSa^.sI_HeadGap.fI_Val / 1000) + fC_HeadOffsetPlate - _pModuleMachineState^.fSubstrateThickness, 1);

// call hardware
(* -- PC PrintController*)
FOR nCtr := 1 TO _nPc DO
  IF _pPc[nCtr] <> 0 THEN
    _pPc[nCtr]^.sI_SystemCmd.bSleep := _iSystemStatus.bSleep;
    _pPc[nCtr]^.sI_SystemCmd.bEStop := _iSystemStatus.bEmergency;
    _pPc[nCtr]^.sI_SystemCmd.bAirNotOk := FALSE;
    _pPc[nCtr]^();
  END_IF
END_FOR

(* -- PH PrintHead*)
FOR nCtr := 1 TO _nPh DO
  IF _pPh[nCtr] <> 0 THEN
    _pPh[nCtr]^();
  END_IF
END_FOR


// Worker
// - fill I_SubSystem correctly from all workers
FOR nCtr := 1 TO GVL_WEU.nC_WorkerPrintPerPm DO
  fbWorkerPrint[nCtr].fPrintStartOffset :=  fPrintOffsetX[nCtr]
                                          + _fDistToMasterPm;
                                  //+ master detect offset,
  fbWorkerPrint[nCtr].bWorkerEnable := _pAdsPm^.bI_Enable AND _pModuleMachineState^.bEngaged AND _pModuleMachineState^.bPrintEnabled;
  fbWorkerPrint[nCtr](
    nPrintPos             := nPos_SubPx,
    bHardwareSync         := bHwSyncCmd,
    bHardwareHold         := FALSE, //bHardwareHold,
    fPrintStartOffset     :=  fPrintOffsetX[nCtr],      // NOTE: dynamic corrections done in Worker (dropSpeedComp / global grid dx / other point corrections))
                            //+ module detect offset,   // modules detect distance or the Master if in simulation mode
                            {warning 'TODO: Vorzeichen von lateral offset & LateralOffser +/-?: Vorher war -'}
    fPrintYOffset         := LIMIT(
                            0,
                                _nYShift_PcRamCenter                      // y-offset for centered image in ph
                                + fPrintOffsetY[nCtr]                     // calc with CB Shift, PU y-Shift, PG y-shift
                                + _pModuleMachineState^.fLateralRegister  // lateral register from machine
                                + _fPrintModuleAdjustY,                   // manual y shift from plc
                            2*_nYShift_PcRamCenter),
    fMasterSpeed          := fSpeed,
    fPUElevation          := fPuElevation,  // for internal dropSpeedCorrection
//    bError                => ,
//    nError                => ,
  );
END_FOR


// machine interface outputs
_pModuleMachineFeedback^.bSpeedExeeded     := checkSpeed(fSpeed:=fSpeed, fMaxSpeed => _pModuleMachineFeedback^.fMaxSpeed);

// messaging
Messaging();

PROPERTY bEngaged : BOOL
GET
bEngaged := _pModuleMachineState^.bEngaged;
END_GET
END_PROPERTY

{attribute 'monitoring':='call'}
PROPERTY bMoving : BOOL
GET
bMoving := _iPrintPosition.bMoving;
END_GET
END_PROPERTY

(* 
  Hardware sync request.
*)
PROPERTY bSyncCmd : BOOL
GET
bSyncCmd := bHwSyncCmd;
END_GET
END_PROPERTY

(*
  Checks if current speed is higher than max. speed.
  :return: TRUE if speed exeeds maximum
*)
METHOD PROTECTED checkSpeed : BOOL
VAR_INPUT
  fSpeed : LREAL;       // current speed
END_VAR
VAR_OUTPUT
  fMaxSpeed : LREAL;    // modules max. printing speed
END_VAR
VAR
  f : LREAL;
  i : UDINT;
END_VAR
VAR_INST
  fbSpeedFilterMav : FB_FILTER_MAV;           // Moving average filter
  fMaxSpeedTolerence : LREAL := 1.0/60;       // Allow max. speed to exeed limit + this tolerance 
END_VAR
// disabled
IF NOT _pAdsPm^.bI_Enable OR NOT _pModuleMachineState^.bEngaged THEN 
  checkSpeed := FALSE;
  fMaxSpeed := 0;
  RETURN;
END_IF 


// filter current speed
fbSpeedFilterMav(fI_Input := fSpeed, iI_NbInputs := 32);  (*max iI_NbInputs = 32!*)

// find slowest max. speed
f := 0;
FOR i:=1 TO GVL_WEU.nC_WorkerPrintPerPm DO
  IF fbWorkerPrint[i].bWorkerEnable THEN
    IF fbWorkerPrint[i].fMaxSpeed = 0 THEN
      ; // ignored speed
    ELSIF f = 0 OR f > fbWorkerPrint[i].fMaxSpeed THEN 
      f := fbWorkerPrint[i].fMaxSpeed;
		END_IF
	END_IF
END_FOR

fMaxSpeed := f;   // return max. possible speed

// check if too fast
IF f > 0 AND fbSpeedFilterMav.fO_OutputMav > f THEN 
  checkSpeed := TRUE; // speed exceeded
ELSE
  checkSpeed := FALSE;
END_IF
END_METHOD

(*
  Distance between activated StartPosition detection and Pm, if one configured (fDetectToCameraOffset + fCameraToPrintOffset)
  If no StartPos detection = 0
*)
PROPERTY fDetectToPm : LREAL
GET
fDetectToPm := fbWorkerCamera.fDetectToCamOffset + fbWorkerCamera.fCameraToPrintOffset;
END_GET
END_PROPERTY

METHOD Init : BOOL
VAR_INPUT
  nIdx                  : UDINT;                                // Module id
  pAdsPm                : POINTER TO ST_ADS_PM;                 // ADS module
  pAdsSa                : POINTER TO ST_ADS_DVTSHEETALIGNMENT;  // ADS sheet alignement
  pAdsCam               : POINTER TO ST_ADS_CAMERA;             // ADS camera
  pAdsPg                : ARRAY[1..GVL_WEU.nC_WorkerPrintPerPm] OF POINTER TO ST_ADS_PG;  // PG -> worker ads 
  
  // config print
  fCycleTime            : LREAL;                // task cycle time in [s]
  fPrintUnitWidth       : LREAL;                // PrintUnit width mechanical [m]
  nYShiftPcCenter       : UDINT;                // Y shift for centered image data in RAM [px]
  // references
  iModuleMaster         : I_ModuleMaster;       // interface for module to master (main) communication
  iPosition             : I_PrintPosition;      // interface for print position
  iStartPos             : I_StartPosDetect;     // interface for start position detect
  iSystemStatus         : I_SystemStatus;       // system status interface (for sleep, estop, ...), may shadow states from machine inputs
  pMachineInputs        : POINTER TO ST_ModuleMachineInterface_IN;
  pMachineOutputs       : POINTER TO ST_ModuleMachineInterface_OUT;
END_VAR
VAR
  nCtr : UDINT;
  sMode : ST_SimModeDef;
END_VAR
IF  pAdsPm = 0 OR pAdsSa = 0 OR pAdsCam = 0 OR 
    pMachineInputs = 0 OR pMachineOutputs = 0 OR
    iModuleMaster = 0 OR iPosition = 0 OR iStartPos = 0 THEN
  LogError('init(): Invalid parameter');
  RETURN;
END_IF

// save config
_nIdx := nIdx;
_pAdsPm := pAdsPm;
_pAdsSa := pAdsSa;
_nYShift_PcRamCenter := nYShiftPcCenter;
_iModuleMaster := iModuleMaster;
_iPrintPosition := iPosition;
_iStartPos := iStartPos;
_iSystemStatus := iSystemStatus;
_pModuleMachineState := pMachineInputs;
_pModuleMachineFeedback := pMachineOutputs;

SetupHw();

// Worker
// -- parameter mediator
fbParamMediator.init(pCamWorker:=ADR(fbWorkerCamera), pDefWorker:=ADR(fbWorkerDeformation));

// -- Worker camera
fbWorkerCamera.Init(iWorkerParams:=iModuleMaster.iWorkerParams, pMsgConfig:=ADR(sL_MsgConfig), fPrintResolution:=_iPrintPosition.fPrintResolution, fSubPxResolution:=_iPrintPosition.fSubPxResolution);
fbWorkerCamera.InitWorkerCamera(pAdsIf:=pAdsCam, iDefGridParamMediator:=fbParamMediator, fPrintUnitWidth:=fPrintUnitWidth);
fbWorkerCamera.reg();
iModuleMaster.registerPuStatusClient(sClient:=fbWorkerCamera);

// -- Worker deformation
fbWorkerDeformation.Init(iWorkerParams:=iModuleMaster.iWorkerParams, pMsgConfig:=ADR(sL_MsgConfig), fPrintResolution:=_iPrintPosition.fPrintResolution, fSubPxResolution:=_iPrintPosition.fSubPxResolution);
fbWorkerDeformation.InitWorkerDeformation(nPrintUnitWidth:=TO_UDINT(F_MeterToSubPixel(fPosMeter:=fPrintUnitWidth, fResoSubPx:=_iPrintPosition.fPrintResolution)), iDefGridParamMediator:=fbParamMediator);
fbWorkerDeformation.reg();
iModuleMaster.registerPuStatusClient(sClient:=fbWorkerDeformation);

// -- Worker print
FOR nCtr := 1 TO GVL_WEU.nC_WorkerPrintPerPm DO
  fbWorkerPrint[nCtr].Init(
    iWorkerParams:=iModuleMaster.iWorkerParams,
    fPrintResolution:=_iPrintPosition.fPrintResolution,
    fSubPxResolution:=_iPrintPosition.fSubPxResolution,
    pMsgConfig:=ADR(sL_MsgConfig)
  );
  fbWorkerPrint[nCtr].InitWorkerPrint(
    pAdsPg:=pAdsPg[nCtr],
    iDefGridParamMediator:=fbParamMediator,
    fLimitCorrectionX:=1000,
    fLimitCorrectionY:=nYShiftPcCenter-1
  );
  fbWorkerPrint[nCtr].reg();
  iModuleMaster.registerPuSubystem(iSubSys:=fbWorkerPrint[nCtr]);
END_FOR 

(*Messaging*)
sL_MsgConfig.bI_Enable       := TRUE;
sL_MsgConfig.pI_FbMsgHandler := ADR(fb_MsgHandler);
fb_MsgHandler.pI_MsgQueue    := ADR(fb_MsgQueue);
fb_MsgQueue.pI_MsgInterface  := ADR(_pAdsPm^.sO_Message);
fb_MsgQueue.cI_MaxElement    := 6;

(*Messages*)
fb_Msg[1].pI_MsgConfig       := ADR(sL_MsgConfig);
fb_Msg[1].iI_MsgLocation     := ePr_BLK_PM;
fb_Msg[1].iI_MsgNumber       := eCMa_COVER_INLET;

fb_Msg[2].pI_MsgConfig       := ADR(sL_MsgConfig);
fb_Msg[2].iI_MsgLocation     := ePr_BLK_PM;
fb_Msg[2].iI_MsgNumber       := eCMa_SECURITY_DOOR_MONITORING;

fb_Msg[3].pI_MsgConfig       := ADR(sL_MsgConfig);
fb_Msg[3].iI_MsgLocation     := ePr_BLK_PM;
fb_Msg[3].iI_MsgNumber       := eCMa_EXHAUST_SYSTEM_WARNING;

fb_Msg[4].pI_MsgConfig       := ADR(sL_MsgConfig);
fb_Msg[4].iI_MsgLocation     := ePr_BLK_PM;
fb_Msg[4].iI_MsgNumber       := eCMa_EXHAUST_SYSTEM_ERROR;

fb_Msg[5].pI_MsgConfig       := ADR(sL_MsgConfig);
fb_Msg[5].iI_MsgLocation     := ePr_BLK_PM;
fb_Msg[5].iI_MsgNumber       := eCMa_EXHAUST_SYSTEM_MALFUNCTION;

fb_Msg[6].pI_MsgConfig       := ADR(sL_MsgConfig);
fb_Msg[6].iI_MsgLocation     := ePr_BLK_PM;
fb_Msg[6].iI_MsgNumber       := eCMa_DRIFT_CONTR_ERROR;

fb_Msg[7].pI_MsgConfig       := ADR(sL_MsgConfig);
fb_Msg[7].iI_MsgLocation     := ePr_BLK_PM;
fb_Msg[7].iI_MsgNumber       := eCMa_AXIS_SAFETY_ACCEPTANCE;

fb_Msg[8].pI_MsgConfig       := ADR(sL_MsgConfig);
fb_Msg[8].iI_MsgLocation     := ePr_BLK_PM;
fb_Msg[8].iI_MsgNumber       := eCPr_SHEET_MARK_DETECTION;

// simulation
sMode.aMode := 'default';
sMode.sCfg  := '{ "desc":"default print module simulation mode" }';
setMode(sMode:=sMode);

bInit := TRUE;
END_METHOD

PROPERTY iPrintPosition : I_PrintPosition
GET
iPrintPosition := _iPrintPosition;
END_GET
END_PROPERTY

PROPERTY iStartPos : I_StartPosDetect
GET
iStartPos := _iStartPos;
END_GET
END_PROPERTY

METHOD PRIVATE Messaging
VAR_INPUT
END_VAR
(*Messaging*)
fb_MsgHandler();

fB_Msg[1](bI_Status := NOT _pModuleMachineState^.bSafetyCoverOk);
fB_Msg[2](bI_Status := NOT _pModuleMachineState^.bServiceDoorsOk);
fB_Msg[3](bI_Status := _pModuleMachineState^.bExhaustVacuumWarning);
fB_Msg[4](bI_Status := _pModuleMachineState^.bExhaustVacuumError);
fB_Msg[5](bI_Status := _pModuleMachineState^.bExhaustFUError);
fB_Msg[6](bI_Status := _pModuleMachineState^.bDriftControlError);
fB_Msg[7](bI_Status := NOT _pModuleMachineState^.bSafetyOk);
fB_Msg[8](bI_Status := _pModuleMachineState^.bDriftControlMissMarks);

fb_MsgQueue();
END_METHOD

(*
  NOTE: Only needed because the Hw instances are outside of the Module.
        Please call the register HW prior initializing the Module itself!
*)
METHOD RegisterHw : BOOL
VAR_INPUT
  pPh : POINTER TO FB_PH_Grid;
  pPc : POINTER TO FB_PC;
  pMapDef : POINTER TO ST_MappingDefinition;
END_VAR
VAR
  i : UDINT;
  bFound : BOOL;
END_VAR
IF pPh = 0 OR pPc = 0 OR pMapDef = 0 THEN LogError('registerHw invalid parameter'); RETURN; END_IF
IF _nPc >= GVL_WEU.nC_MaxPcPerPm THEN LogError('register hw: too many PCs registered'); RETURN; END_IF
IF _nPh >= GVL_WEU.nC_MaxPhPerPm THEN LogError('register hw: too many PHs registered'); RETURN; END_IF

// PC 
bFound := FALSE;
FOR i:=1 TO _nPc DO   // search for existing pc
  IF _pPc[i] = pPc THEN bFound := TRUE; EXIT; END_IF
END_FOR
IF NOT bFound THEN    // add if unknown
  _nPc := _nPc + 1;
  _pPc[_nPc] := pPc;
  _nPcToWorker_Mapping[_nPc] := pMapDef^.nPg;  // save mapping
ELSE
  ; // ignore new pc
END_IF

// PH
bFound := FALSE;
FOR i:=1 TO _nPh DO   // search for existing ph
  IF _pPh[i] = pPh THEN bFound := TRUE; EXIT; END_IF
END_FOR
IF NOT bFound THEN    // add if unknown
  _nPh := _nPh + 1;
  _pPh[_nPh] := pPh;
  _nPhToPc_Mapping[_nPh] := pMapDef^.nPc;
  _nPhToPcCh_Mapping[_nPh] := pMapDef^.nPcCh;
  _nPhToWorker_Mapping[_nPh] := pMapDef^.nPg;
ELSE
  LogWarning(F_Concat3('FB_PH=', pPh^.sName, ', already registered, ignore'));
END_IF

RegisterHw := TRUE;
END_METHOD

METHOD PROTECTED setLogLevels
VAR_INPUT
  lvl : E_LogSeverity;
END_VAR
// set logging levels
fbWorkerCamera.LogLevel := lvl;
fbWorkerPrint[1].LogLevel := lvl;
fbWorkerPrint[2].LogLevel := lvl;
END_METHOD

(*
  Links hw to mapped handlers.
  NOTE: override this method if it does not match the default mapping.
*)
METHOD PRIVATE SetupHw
VAR
  i : UDINT;
END_VAR
IF _iModuleMaster.iHardwarePool = 0 THEN LogError('SetupHw: invalid hw pool reference, do not setup'); RETURN; END_IF
// PC
FOR i := 1 TO _nPc DO
  IF _pPc[i] = 0 THEN LogError(F_Concat4('SetupHw: invalid pc mapping','_pPc[',TO_STRING(i),']=0'));
    CONTINUE;
	END_IF

  // register to worker
  fbWorkerPrint[_nPcToWorker_Mapping[i]].registerPc(iNewPC:=_pPc[i]^);
  
  // register to hw pool
   _iModuleMaster.iHardwarePool.registerPc(pNewPc:=_pPc[i]);
END_FOR

// PH
FOR i := 1 TO _nPh DO
  IF _pPh[i] = 0 OR _pPc[_nPhToPc_Mapping[i]] = 0 THEN LogError(F_Concat4('SetupHw: invalid ph mapping','_pPh[',TO_STRING(i),']=0'));
    CONTINUE;
	END_IF
  
  // register to worker
  fbWorkerPrint[_nPhToWorker_Mapping[i]].registerPh(iPH:=_pPh[i]^, iNewCG:=_pPh[i]^);
  
  // register to hw pool
  _iModuleMaster.iHardwarePool.registerPh(pNewPh:=_pPh[i]);
  
  // link ph <-> pc if not done externally
  _pPc[_nPhToPc_Mapping[i]]^.registerPH(iPH :=_pPh[i]^, nCh := TO_UINT(_nPhToPcCh_Mapping[i]));

END_FOR
END_METHOD

END_FUNCTION_BLOCK

// ---- POUs/Products/Print_Weu/FB_WorkerDefGrid_Print_WEU.TcPOU
FUNCTION_BLOCK FB_WorkerDefGrid_Print_WEU EXTENDS FB_WorkerDefGrid IMPLEMENTS I_PrintSubsystem
VAR_INPUT
  nPrintPos             : DINT;   // Absolute printing position [SubPx]
  fMasterSpeed          : LREAL;  // Speed [m/s]
  bHardwareSync         : BOOL;   // hw sync signal (chenerates a triger internally)
  bHardwareHold         : BOOL;   // hw hold signal
  fPrintStartOffset     : LREAL;  // X-Shift StartOffset from Module reference (configurative PU/PM/PG/PA ADS offset) [m]
  fPrintYOffset         : LREAL;  // Y-Shift
  // correction live parameter
  fPUElevation          : LREAL;  // PU distance from substrate [m]
END_VAR
VAR
  // print
  // - references
  _pAdsPg            : POINTER TO ST_ADS_PG;      // pg ads reference (for pa)
  // - instances
  fbPs               : FB_PS_Grid;
  fbPa               : FB_PA;
  fB_PcAdapter       : FB_PC_Adapter;
  
  // grid specific
  // - references
  _iParamMediator    : I_ParamMediator;
  // - settings
  sDefGridSettings   : ST_DefGridSettings; 
  // - state 
  fCurrentColumnPos  : LREAL; // Currently column position
  fCurrentPreCharge  : LREAL; // Currently to be precharged
  nChargedColumns    : UDINT; // Already charged columns


  // print corrections
  nPointCorrections  : UDINT;     // number of registered point correction handler
  iPointCorrections  : ARRAY[1..nC_NUM_POINTCORRECTIONS] OF I_GridPointCorrection;  // point corrections
  
  // - Time of flight correction of droplets
  fbDropSpeedComp    : FB_DropSpeedComp;
  //
  _pAdsCam           : POINTER TO ST_ADS_CAMERA;  // camera interface PUC
  // - global shifts (applied globally and not on every single point (calcualted based on all CT points))
  _fDxGlobalShift    : LREAL;
  _fDyGlobalShift    : LREAL;

  // settings or helper
  _fPrintStartOffset : LREAL;   // internal print start offset (distance Cam -> PG1 + PG Offset + PU offset)
  _nPosX0            : DINT;    // X0 for last attached CT (detected postion)
  _nPosXS            : DINT;    // XS for last attached CT (shifted print start position)
  _nPosXDelta        : DINT;    // Shift value X0 -> XS
  _fPosY             : LREAL;   // Y shift for last attached CT
  _nPosDeltaToPrint  : DINT;    // delta pos in [SbuPx] from attach to print
  _sCurrentImgDepth  : LREAL;   // Job: current image length [m]
  _bEndless          : BOOL;    // Job: endless
  _bPaStarted        : BOOL;
  _bPaStartRequested : BOOL;
  _sJobDef           : BOOL;
  fBStartTimeout     : TON;
  rTrigHwSync        : R_TRIG;
  _bForceDefGridOff  : BOOL;    // force deformation grid stream to ph off (send 0)
  
  (*grid limit*)
  _fLimitCorrectionX : LREAL;     // correction limit in y (abs) [px]
  _fLimitCorrectionY : LREAL;     // correction limit in y (abs) [px]
    
  (*Messaging*)
  (*we could implement a message handler for ST_ADS_PG message interface*)

END_VAR

VAR PERSISTENT
  _fColumnsToPrecharge : LREAL := nC_COLUMNS_TO_PRECHARGE;
  _fStartShiftOffset   : LREAL := fC_START_SHIFT_OFFSET;
  _fStartShiftFactor   : LREAL := fC_START_SHIFT_FACTOR;
END_VAR

VAR CONSTANT
  iC_NUM_MSG               : UDINT := 5;
  nC_COLUMNS_TO_PRECHARGE  : LREAL := 2.1;
  fC_GRIDPOINT_STREAM_TIME : LREAL := 0.0025;     // time to stream one point [s]
  fC_START_SHIFT_FACTOR    : LREAL := -2.4E-2;
  fC_START_SHIFT_OFFSET    : LREAL := -1.0E-2;
  nC_NUM_POINTCORRECTIONS  : UDINT := 5;
END_VAR

(*
DOC:
What will be different to FB_WorkerDefGrid_Print of DMAX
- Re-Sync StartPosDetect interface with optional camera data (y-shift)
  Clear with Attach(), security clearance
- (maybe not needed) Stream grid faster to PC (we have no break for switching the CT in endless)
- New PDI StartPostion update (+print start only for first CT) --> send to NIOS or hw buffer
- PDI GridPoint stream
- New PDI PrintingLength update (after last streamed point)
- Other rules for Worker position calculation
*)

PROPERTY aPaState : STRING
GET
aPaState := fbPa.aPaState;
END_GET
END_PROPERTY

METHOD PROTECTED  Attach : BOOL
VAR_INPUT
  iCT              : I_CT;                         (*container at triggered event position*)
END_VAR
Attach:=FALSE;

IF SUPER^.Attach(iCT:=iCT) THEN
  // Additional worker checks
    // - job is valid?
  IF _pAttachedCt^.pJob = 0 OR NOT _bJobActive THEN
    Release(iCT:=iCT);
    RETURN;   // do not print
  
  // CT valid & CT present
  ELSIF NOT _pAttachedCt^.bValid OR NOT _pAttachedCt^.bProductPresent THEN
    Release(iCT:=iCT);
    RETURN;   // do not print
  
  // Ignore start due to hardware hold  
  ELSIF bHardwareHold THEN
    _pAttachedCt^.setError(ErrDef:=EC_Print.ecPaAbortHold, Src:=_pEcSrc^);
    Release(iCT:=iCT);
    RETURN;   // do not print
  
  // - OK attach
  ELSE
    Attach := TRUE;
	END_IF
  
  
  //Prepare print station
  sDefGridSettings := _iParamMediator.sDeformationGridSetttings; // or get from CT (but needs to be set even if WorkerDeformation is not enabled) _pAttachedCt^.sDefGridSettings;
  // fix some potential errors
  IF sDefGridSettings.nGridPitchX = 0 THEN sDefGridSettings.nGridPitchX :=1024; LogError(F_concat2('grid not configured, set default nGridPitchX=',TO_STRING(sDefGridSettings.nGridPitchX))); END_IF
  IF sDefGridSettings.nGridPitchY = 0 THEN sDefGridSettings.nGridPitchY :=1024; LogError(F_concat2('grid not configured, set default nGridPitchY=',TO_STRING(sDefGridSettings.nGridPitchY))); END_IF
  
  nChargedColumns := 0;
  fbPs.bPrintEnable := iCT.bValid AND iCT.bProductPresent;
  fbPs.setGrid(sGrid:=sDefGridSettings);
  _fDxGlobalShift := _pAttachedCt^.fDxShift;
  _fDyGlobalShift := _pAttachedCt^.fDyShift;

  //Start print, PA should be in READY or DONE
  
  // Set X print position
  _nPosX0 :=    _pAttachedCt^.getPosX0(nPosDomain:=E_PosDomain.master_pos)
              //- General Shift
              - F_MeterToSubPixel(fbDropSpeedComp.fDropPlacementError, _fPrintResolution*_fSubPxResolution); // - drop compensation*)
  _nPosXDelta := F_MeterToSubPixel(_fPrintStartOffset, _fPrintResolution*_fSubPxResolution); // + PG/PA Shift (additional PG offset 0 for firstLine)
  
  IF GVL_Deformation.bC_UseGlobalGridShift THEN
    _nPosXDelta := _nPosXDelta + FC_LREAL_TO_DINT(_fDxGlobalShift);                  // + global shift from grid points
  END_IF

  _nPosXS := _nPosX0 + _nPosXDelta;
  fB_PcAdapter.setPrintStartPos(nX0:=_nPosXS);
  
  // Set Y print position
  _fPosY := fPrintYOffset;
  IF GVL_Deformation.bC_UseGlobalGridShift THEN
    _fPosY := _fPosY + _fDyGlobalShift;    // + global shift from grid points
  END_IF
  fB_PcAdapter.setPrintYShift(nYShift:=FC_LREAL_TO_DINT(_fPosY));

  // check
  IF _nPosXS < nPrintPos THEN
    LogWarning(Msg:=F_Concat4('Print start position:', TO_STRING(_nPosXS) ,' < Encoder position:', TO_STRING(nPrintPos)));
	END_IF
  
  // save current distance to print position
  _nPosDeltaToPrint := _nPosXS - iCT.GetPos(nPosDomain:=E_PosDomain.master_pos) - _nPosX0;
  checkGridTiming();
  
  
  IF NOT fbPa.bPrinting THEN   // fB_PcAdapter.bAllPrinting
    IF NOT fbPa.printStart() THEN
      LogError(Msg:='PA not ready to start at attach');
      Release(iCT := iCT);
    ELSE
      _bPaStarted := FALSE;
      _bPaStartRequested := TRUE;
      Attach:=TRUE;
    END_IF
  ELSE
    // update start postion if it was already started (endless)
    {warning 'TODO: implement print restart in endless'}
    //fbPa.restartPrint();
    Attach:=TRUE;
  END_IF
  
  // debug log
  LogLvl(Lvl:=E_LogSeverity.Debug, F_Concat4('printStart: at XS:', TO_STRING(_nPosXS), ' ', _pAttachedCt^.print(0)));  // print container
  IF GVL_Deformation.bC_UseGlobalGridShift THEN
    LogLvl(Lvl:=E_LogSeverity.Debug, F_Concat4(
                                        F_Concat3('> XS = X0(', TO_STRING(_pAttachedCt^.GetPosX0(nPosDomain:=E_PosDomain.master_pos)), ')'),
                                        F_Concat3(' + shDx(', TO_STRING(_fDxGlobalShift), ')'),
                                        F_Concat3(' + shStartOffs(', TO_STRING(F_MeterToSubPixel(_fPrintStartOffset,_fPrintResolution*_fSubPxResolution)), ')'),
                                        F_Concat3(' - shDropComp(', TO_STRING(F_MeterToSubPixel(fbDropSpeedComp.fDropPlacementError,_fPrintResolution*_fSubPxResolution)), ')')
                                     ));
  ELSE
    LogLvl(Lvl:=E_LogSeverity.Debug, F_Concat3(
                                        F_Concat3('> XS = X0(', TO_STRING(_pAttachedCt^.GetPosX0(nPosDomain:=E_PosDomain.master_pos)), ')'),
                                        F_Concat3(' + shStartOffs:', TO_STRING(F_MeterToSubPixel(_fPrintStartOffset,_fPrintResolution*_fSubPxResolution)), ')'),
                                        F_Concat3( ' - shDropComp:', TO_STRING(F_MeterToSubPixel(fbDropSpeedComp.fDropPlacementError,_fPrintResolution*_fSubPxResolution)), ')')
                                     ));
  END_IF
  
  
ELSE
  // parent attach failed case
END_IF
END_METHOD

PROPERTY bPausePrintCanEx : BOOL
GET
bPausePrintCanEx := FALSE; //Not implemented
END_GET
END_PROPERTY

PROPERTY bPcEnabled : BOOL
GET
bPcEnabled := fB_PcAdapter.bPcEnable;
END_GET
END_PROPERTY

PROPERTY bPrintEnabled : BOOL
GET
bPrintEnabled := _bEnable;
END_GET
END_PROPERTY

PROPERTY bPrintError : BOOL
GET
bPrintError := bError; // Worker error 
                  // or fB_PcAdapter.bError
END_GET
END_PROPERTY

PROPERTY bPrinting : BOOL
GET
bPrinting := fbPa.bPrinting;
END_GET
END_PROPERTY

PROPERTY bPrintReady : BOOL
GET
bPrintReady := fbPa.bReady;
END_GET
END_PROPERTY

PROPERTY bStartPrintCanEx : BOOL
GET
bStartPrintCanEx := fbPa.bStartCanEx;
END_GET
END_PROPERTY

PROPERTY bStopPrintCanEx : BOOL
GET
bStopPrintCanEx := fbPa.bStopCanEx;
END_GET
END_PROPERTY

{attribute 'monitoring':='call'}
PROPERTY bWorkerEnable : BOOL
GET
bWorkerEnable := SUPER^.bWorkerEnable;
END_GET
SET
IF _pAdsPg = 0 THEN
  SUPER^.bWorkerEnable := bWorkerEnable;
ELSE
  // mask worker enable with group enable
  SUPER^.bWorkerEnable := bWorkerEnable AND _pAdsPg^.bI_Enable;  
END_IF
END_SET
END_PROPERTY

METHOD PRIVATE checkGridTiming : BOOL
VAR
END_VAR
// check for timing problems
IF fMasterSpeed <> 0 THEN

  // - check pre-charge at beginning
  IF _fColumnsToPrecharge * fC_GRIDPOINT_STREAM_TIME * GVL_Deformation.nC_GridRoiRows >= F_SubPixelToMeter(lPosSubPx:=_nPosDeltaToPrint, fResSubPx:=_fPrintResolution*_fSubPxResolution) / fMasterSpeed  THEN
       LogError('Machine too fast for grid stream (for pre-charge at attach)');
  END_IF
  
 // - check charge time needed per columns vs machine speed and grid-sizeY
 IF GVL_Deformation.nC_GridRoiRows * fC_GRIDPOINT_STREAM_TIME >= F_SubPixelToMeter(lPosSubPx:=TO_DINT(sDefGridSettings.nGridPitchX), fResSubPx:=_fPrintResolution) / fMasterSpeed THEN
   LogError('Machine too fast for grid stream (time rows per column)');
 END_IF

END_IF
END_METHOD

(*
  Limit correction to boundaries
  :return: TRUE if limited
*)
METHOD PRIVATE correctionLimit : BOOL
VAR_INPUT
  pPoint : POINTER TO ST_DeformationPointAccurate;
END_VAR
VAR
  bLimited : BOOL;
  nExeedX, nExeedY : LREAL;
END_VAR
// limit point correction to boundaries and inform
IF    pPoint^.dx >= _fLimitCorrectionX    THEN nExeedX := pPoint^.dx; pPoint^.dx := _fLimitCorrectionX;    bLimited:=TRUE; 
ELSIF pPoint^.dx <= -1*_fLimitCorrectionX THEN nExeedX := pPoint^.dx; pPoint^.dx := -1*_fLimitCorrectionX; bLimited:=TRUE;
ELSIF pPoint^.dy >= _fLimitCorrectionY    THEN nExeedY := pPoint^.dy; pPoint^.dy := _fLimitCorrectionY;    bLimited:=TRUE;
ELSIF pPoint^.dy <= -1*_fLimitCorrectionY THEN nExeedY := pPoint^.dy; pPoint^.dy := -1*_fLimitCorrectionY; bLimited:=TRUE;
END_IF
IF bLimited THEN 
  LogLvl(Lvl:=E_LogSeverity.Warning, Msg:=F_Concat5( 'Point=',TO_STRING(pPoint^.index),
                                                     F_Concat5(' c/r(',TO_STRING(pPoint^.col),'/',TO_STRING(pPoint^.row), ') '),
                                                     F_Concat4('dx:', TO_STRING(nExeedX), ' dy:', TO_STRING(nExeedY)),
                                                     ' correction exceeded limit')); 
END_IF
correctionLimit := bLimited;
END_METHOD

METHOD PRIVATE correctionUpdate : BOOL
VAR_INPUT
  pPoint : POINTER TO ST_DeformationPointAccurate;
END_VAR
VAR
  i : UDINT;
END_VAR

// here apply all PU specific corrections
// - mechanical stretch based on temperature extension (if not done in Camera)
// - banana correction
// - Y-shifts of PU
// - trapzedoial correction
// - ...

// global dx/dy correction
//   remove global shift from GridPoints (shifted by PU)
IF GVL_Deformation.bC_UseGlobalGridShift THEN
  pPoint^.dx := pPoint^.dx - _fDxGlobalShift;
  pPoint^.dy := pPoint^.dy - _fDyGlobalShift;
END_IF

// PU Deformation correction
IF GVL_Deformation.bC_UsePUDeformation THEN
  FOR i:=1 TO nPointCorrections DO
    iPointCorrections[i].updateCorrection(pPoint:=pPoint);
  END_FOR
END_IF
END_METHOD

(*
  Max. supported speed [m/s], 0 if not available
*)
{attribute 'monitoring':='call'}
PROPERTY fMaxSpeed : LREAL
GET
VAR
  nSpeedMpMin : DINT;
END_VAR
nSpeedMpMin := SEL(bWorkerEnable AND _pAdsPg <> 0, 0, _pAdsPg^.sI_MaxPrintSpeed.lI_Val);
fMaxSpeed := TO_LREAL(nSpeedMpMin)/60;
END_GET
END_PROPERTY

{attribute 'monitoring':='call'}
PROPERTY fStartShiftFactor : LREAL
GET
fStartShiftFactor := _fStartShiftFactor;
END_GET
SET
_fStartShiftFactor := fStartShiftFactor;
END_SET
END_PROPERTY

{attribute 'monitoring':='call'}
PROPERTY fStartShiftOffset : LREAL
GET
fStartShiftOffset := _fStartShiftOffset;
END_GET
SET
_fStartShiftOffset := fStartShiftOffset;
END_SET
END_PROPERTY

METHOD PROTECTED gridUpdate : BOOL
VAR_INPUT
  bEnableDeformation : BOOL;      // enable correction update, else correction (0/0) is written
END_VAR
VAR
  sPoint : ST_DeformationPointAccurate;
  nRow : UDINT;
  nAvailPoints : UDINT;
  nConvErr : UDINT;
END_VAR
VAR_INST
  nAvailPoints_mem : UDINT;
END_VAR
//TODO: rewrite this method to look cleaner (less if else)
IF sDefGridSettings.nGridSizeX = 0 THEN RETURN; END_IF          // avoid endless loops
IF sDefGridSettings.nGridSizeY = 0 THEN RETURN; END_IF

gridUpdate:=TRUE;

// calculate grid column position
IF sDefGridSettings.nGridPitchX <> 0 THEN
  fCurrentColumnPos := fCtPosition / (sDefGridSettings.nGridPitchX * _fSubPxResolution);   // calc grid column position relative to worker
END_IF

